	machineStates.stStartUp:
		Global.emgStop       := FALSE;
		Global.openDoors     := FALSE;
		Global.emgStopSignal := FALSE;
		resetSig             := FALSE;
		commandReady         := FALSE;
		purgeIndexDone       := FALSE;
		purgeRobotDone       := FALSE;
		purgeStackers		 := FALSE;
		Global.commands      := controlCommands.null;
		setDisplayState(machineDisplayStates.dStStartUp);
		NextState(machineStates.stInit);
	
//  *** Safety stop 
//  Има отворена врата, няма въздух или има натисната губа
//  Към всички станций се подава EMG сигнал

	machineStates.stSafetyStop:
		Global.commands      := controlCommands.null;
		Global.emgStopSignal := TRUE;
		resetTimer(IN := resetSig, PT := resetTime);
		
		IF      io.getX(ioImage.xDoors) 
			AND io.getX(ioImage.xAirOk) 
			AND io.getX(ioImage.xEmgBnt) 
			AND io.getX(ioImage.xRobotEmgOk)  THEN
				resetSig := TRUE;
				IF resetTimer.Q THEN	
					resetSig      := FALSE;
					nextState(machineStates.stInit);
				END_IF
		END_IF	

//  *** Init 
//  Инициализация на всички станций 
			
	machineStates.stInit:
		setDisplayState(machineDisplayStates.dStMachineStandBy);
		
		CASE Global.commands OF	
			controlCommands.start, 
			controlCommands.stop:
		        commandReady         := TRUE;
				Global.machError     := FALSE;
			    Global.emgStopSignal := FALSE;
			    nextState(machineStates.stReady);
				
			    Stations.incCommStBase.DoInit      := TRUE;			
			    Stations.sLoadStBase.DoInit        := TRUE;
				Stations.sUnloadStBase.DoInit      := TRUE;
				Stations.insertLoadStBase.DoInit   := TRUE;
				Stations.insertUnloadStBase.DoInit := TRUE;				
				Stations.roboStBase.DoInit         := TRUE;		
			
		END_CASE

// *** Ready 
// Синхронизира всички станций след подаване на захранването

	machineStates.stReady:
		depSync(Stations.incCommStBase,      globalDeps.depIncCommModeDone); 
		depSync(Stations.sLoadStBase,        globalDeps.depSLoadInit);
		depSync(Stations.sUnloadStBase,      globalDeps.depSUnloadInit);
		depSync(Stations.insertLoadStBase,   globalDeps.depILoadInitDone);
		depSync(Stations.insertUnloadStBase, globalDeps.depULoadInitDone);
		depSync(Stations.roboStBase,         globalDeps.depRoboInitDone);	
	
		nextState(machineStates.stCheckState);	
		
// *** Check state 
// В зависимост от зададената команда се задава следващо състояние

	machineStates.stCheckState:	
		IF NOT Global.purgeActive THEN	
			
			CASE Global.commands OF	
				controlCommands.start:
					nextState(machineStates.stAutoRun);
		   		controlCommands.stop:		
					nextState(machineStates.stStopping);
			END_CASE
			
		ELSE
			// Активна е purge процедура
			// Изчаква да се изпразни масата
			IF NOT purgeIndexDone THEN
				nextState(machineStates.stPurgeDialIndexSync);
			END_IF
			
			// Изчаква робота на приключи работа
			IF NOT purgeRobotDone THEN
				nextState(machineStates.stPurgeRobot);
			END_IF		

			// Изчаква стакерите да изкарат тарите в тях
			IF NOT purgeStackers THEN
				nextState(machineStates.stPurgeStackers);
			END_IF	
			
			nextState(machineStates.stPurgeDone);
			
		END_IF	

//  *** Stopping
//  Изчакват се всички станций да спрат

	machineStates.stStopping:
		setDisplayState(machineDisplayStates.dStMachineIsStopping);
		depSignal(globalDeps.depMachineStopping);
		depSync(Stations.incCommStBase,      globalDeps.depIncStop);		
		depSync(Stations.sLoadStBase,        globalDeps.depSLoadStop);
		depSync(Stations.sUnloadStBase,      globalDeps.depSUnloadStop);
		depSync(Stations.insertLoadStBase,   globalDeps.depILoadStop);
		depSync(Stations.insertUnloadStBase, globalDeps.depULoadStop);
		depSync(Stations.roboStBase,         globalDeps.depRoboStop);
		
		nextState(machineStates.stStopMach);
		
//  *** Stop 
//  Машината е спряна

	machineStates.stStopMach:	
		IF commandReady THEN
			Global.commands    := controlCommands.null;
			commandReady       := FALSE;	
		END_IF
	    setDisplayState(machineDisplayStates.dStMachineIsStopped);
	  
	    CASE Global.commands OF	
	      controlCommands.start:
		  	 commandReady := TRUE;
			 IF NOT Global.purgeActive THEN
		  		 nextState(machineStates.stAutoRun);	
			 ELSE
		  		 nextState(machineStates.stPurgeStart);
			 END_IF				 
							
		END_CASE	
	  
//  *** Auto run
//  Автоматичен режим

	machineStates.stAutoRun:
		IF commandReady THEN
			Global.commands    := controlCommands.null;
	    	commandReady       := FALSE;	
		END_IF
	    setDisplayState(machineDisplayStates.dStAutoRun);
		depSignal(globalDeps.depMachineAuto);
		IF Global.commands = controlCommands.stop THEN
		  	 commandReady := TRUE;				
		  	 nextState(machineStates.stStopping);			
		END_IF

// *** Purge - Start
// Изчистване на останалите в машита бройките
	
	machineStates.stPurgeStart:
		purgeIndexDone       := FALSE;
		purgeRobotDone       := FALSE;
		purgeStackers		 := FALSE;
		setDisplayState(machineDisplayStates.dStMachinePurgeActive);
		depSignal(globalDeps.depMachinePurgeStart);
		nextState(machineStates.stPurgeDialIndexSync);	
		
// *** Purge - Dial Index Sync
// Изчаква масата на InC да се завърти колкое необходимо пъти
// зада се изчистят останалите броки от нея
	
	machineStates.stPurgeDialIndexSync:	
		purgeIndexDone := FALSE;
		depSync(Stations.incCommStBase, globalDeps.depIncPurgeDone);
		nextState(machineStates.stPurgeRobot);		
		
// *** Purge - Robot Start
// Команда purge към робота
	
	machineStates.stPurgeRobot:	
		purgeIndexDone := TRUE;
		purgeRobotDone := FALSE;
		depSignal(globalDeps.depMachinePurgeRobot);
		depSync(Stations.roboStBase, globalDeps.depRoboPurgeDone);
		nextState(machineStates.stPurgeStackers);
		
// *** Purge - Stackers
// Команда purge към стакерите
	
	machineStates.stPurgeStackers:
		purgeRobotDone := TRUE;
		purgeStackers  := FALSE;	
		depSignal(globalDeps.depMacinePurgeStackers);	
		depSync(Stations.sLoadStBase,   globalDeps.depSLoadPurgeDone);	
		depSync(Stations.sUnloadStBase, globalDeps.depSUnloadPurgeDone);	
		nextState(machineStates.stPurgeDone);

// *** Purge - Done

	machineStates.stPurgeDone:	
		purgeStackers		 := TRUE;
		Global.purgeActive   := FALSE;
	    TagsHMI.startPurge   := FALSE;		
		nextState(machineStates.stStop);				
	
//  *** Machine error
//  В някоя станция има грешка

	machineStates.stMachError:
		Global.commands    := controlCommands.null;
		setDisplayState(machineDisplayStates.dStStationError);		
	
END_CASE

METHOD PRIVATE setEmg
VAR_INPUT
	
	emgOrAlarm				: Bool; 				// Дали метода е извикам за EMG stop или аларма

END_VAR

// Когато има EMG ситуация или аларма, се задава съответният state, 
// без оглед на текущото състояние на state машината.
// Аварийното спиратен е с по-голям приоритет от алармата

	stBase.DependencyState       := Consts.NO_DEPENDENCY;
	depActive                    := FALSE;
	syncActive                   := FALSE;
	statePass 			   		 := FALSE;
	depCount                     := 0;
	MEMSET(ADR(syncArr), 0, SIZEOF(syncArr));
	
	IF emgOrAlarm THEN
		stCurrentState               := machineStates.stSafetyStop;
		stBase.CurrentState          := machineStates.stSafetyStop;
	ELSE
		stCurrentState               := machineStates.stMachError;
		stBase.CurrentState          := machineStates.stMachError;
	END_IF
END_METHOD

ACTION zumer:
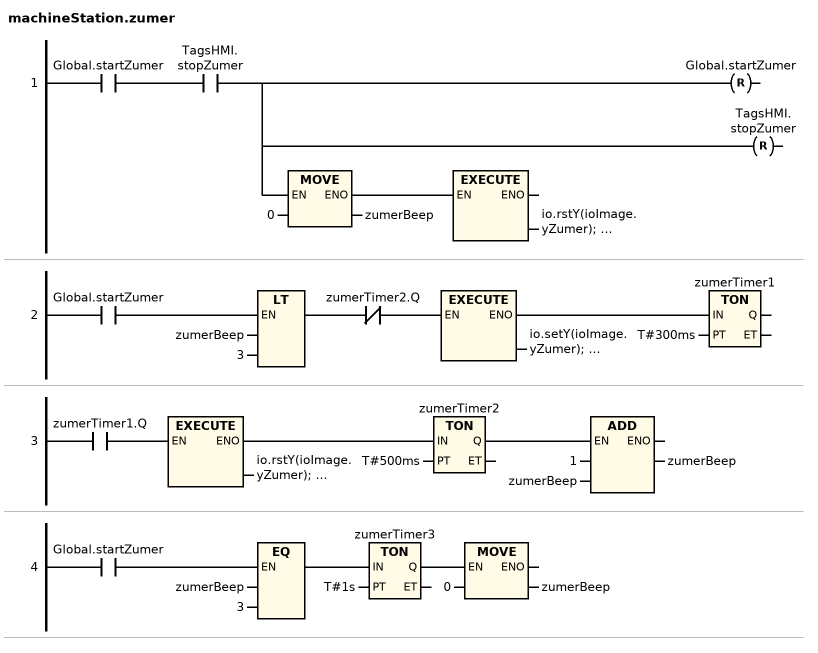
// NETWORK 1
_w1 := Global.startZumer AND TagsHMI.stopZumer;
Global.startZumer R= _w1;
TagsHMI.stopZumer R= _w1;
IF _w1 THEN zumerBeep := 0; END_IF
IF _w1 THEN io.rstY(ioImage.yZumer); END_IF

// NETWORK 2
_w2 := (Global.startZumer AND zumerBeep < 3) AND NOT zumerTimer2.Q;
IF _w2 THEN io.setY(ioImage.yZumer); END_IF
zumerTimer1(IN := _w2, PT := T#300ms); // TON

// NETWORK 3
_w3 := zumerTimer1.Q;
IF _w3 THEN io.rstY(ioImage.yZumer); END_IF
zumerTimer2(IN := _w3, PT := T#500ms); // TON
IF zumerTimer2.Q THEN zumerBeep := 1 + zumerBeep; END_IF

// NETWORK 4
zumerTimer3(IN := Global.startZumer AND zumerBeep = 3, PT := T#1s); // TON
IF zumerTimer3.Q THEN zumerBeep := 0; END_IF
END_ACTION

END_FUNCTION_BLOCK

// ---- POUs/stateMachine.TcPOU
FUNCTION_BLOCK stateMachine
VAR_INPUT

	stBase             : REFERENCE TO stationBase;	// Базова структура на станция  
	activeEMG          : BOOL;                      // Има активен safety стоп
	
	depClear           : BOOL;
	syncClear          : BOOL;

	
	
END_VAR
VAR_OUTPUT
END_VAR


VAR
	stCurrentState     : DINT;  			        // Текущо състояние на станцията
	startUp            : BOOL := FALSE;    		    // Флаг който се сетва за 1 цикъл при първо извикване 
	statePass		   : BOOL; 						// Вече има избран следващ state
	depPass            : BOOL; 						// Depandancy е било изпълнено за даденият state
	depSyncPass		   : BOOL;                    // Всички завицещи от текущият state, други станций са били sync-нати
	stationStop		   : BOOL; 				        // Станцията е спряна
	depActive          : BOOL;                      // Станцията изчаква друга
	syncActive         : BOOL;                      // Станцията sync-ва друга
	syncArr            : ARRAY [0..Consts.MAX_SYNC_STATIONS] OF INT; 
	depCount           : INT;                       // Общ брой на dependency-ta към други станий в текущият state
	depIndex           : INT;                       // Индек за адресиране на dependency в syncArr
	stTimer		       : TON;						// Всяки state има по един таймер
	stErrTimer         : TON;                       // И по един за генериране на грешка 
	startTimer         : BOOL;                      // Битове за старт на таймерите
	startErrTimer      : BOOL;
	stTime             : TIME;                      // Време на stTimer-a - задава се от stаteDalay
	stErrTime          : TIME;                      // Време за stErrТimer-a - задава се от timeOutError
	io				   : ioControl;                 // Дефинира няколко метода за работа с IO
	tempState          : DINT;                      // Запазва некущото състояни за step mode
	stepModeActive     : BOOL; 						// Активен е стъпков режим
	debugTimer         : TON;
	debugTImerIN       : BOOL;

END_VAR


// Тази част на FB-то никога няма да се изпълни (и кода в нея)

METHOD PRIVATE cycle
VAR_INPUT
	
	ioImage            : ANY;                           // ioImage за станцията 
	
END_VAR

VAR 
	ioImageIndex    : POINTER TO DINT;                 // показва началото на IO Image структурата
	ioStruct		: POINTER TO imageIO;              // текуща структура - една IO точка (DI или DO)
	points 			: DINT;							   // брой на входове и изходи в дадената стация
END_VAR

// Служи за упр. на стъпковата машина (в случея Switch Case блок)
// Грижи се за правилното упр. на сигнали от Staion Base

// Станцията е на автоматичен режим и е активна
IF stBase.AutoMode AND stBase.ToggleEnable THEN
	
	stBase.Disabled := FALSE;
	
	// Индекса за dependency-та се нулара всеки цикъл (изпползва се в dependencySync)
	depIndex        := 0;
		
	// При първо извикване станцията преминава в стартово състояние
	IF NOT startUp THEN
		startUp 			 	   	 := TRUE;
		stBase.Busy 	      	 	 := FALSE;
		stBase.Ready		 	 	 := FALSE;
		stBase.Error    	  		 := FALSE;
		stBase.LastState      		 := Consts.ST_START_UP;
		stBase.CurrentState   		 := Consts.ST_START_UP;
		stBase.Error          		 := FALSE;
		stBase.LastErrorState        := Consts.ST_NULL;
		stBase.DoInit         		 := FALSE;
		stBase.DoStart        		 := FALSE;
		stBase.DoStop        		 := FALSE;
		stBase.DependencyState       := Consts.NO_DEPENDENCY;	
		stCurrentState 				 := Consts.ST_START_UP;
		tempState 				     := Consts.ST_NULL;
		depCount 				     := 0;
		depActive                    := FALSE;
		syncActive                   := FALSE;
		statePass 			   		 := FALSE;
		depPass 				     := FALSE;
		depSyncPass 			     := FALSE;
		MEMSET(ADR(syncArr), 0, SIZEOF(syncArr));

	END_IF
	
	// Без оглед на текущото състояние се задава състояние на стоп
    // Ако има започанала някаква манупулация тя ще завърши 

	IF stBase.DoStop THEN
	
		stBase.DoStop             := FALSE;
		stationStop               := TRUE; 
		stBase.Busy 	      	  := FALSE;
		stBase.Ready		 	  := FALSE;
		stBase.Error              := FALSE;
		stepModeActive            := FALSE;
		depCount 				  := 0;
		depActive                 := FALSE;
		syncActive                := FALSE;
		statePass 			      := FALSE;
		depPass 				  := FALSE;
		depSyncPass 			  := FALSE;		
		stBase.CurrentState       := Consts.ST_STOP;
		tempState 				  := Consts.ST_NULL;
	
	END_IF
	
	// Когато станцията е спряла или е имало грешка при командта RESTART от HMI (DoInt)
	// станцията се инициализира
	IF  stBase.DoInit THEN
		
	    stBase.DoInit                := FALSE;
		stBase.Error                 := FALSE;
		stationStop    			     := FALSE;
		statePass 			   		 := FALSE;
		stBase.DoConfirmDependency   := FALSE;
		depCount 				     := 0;
		depActive                    := FALSE;
		syncActive                   := FALSE;
		statePass 			   		 := FALSE;
		depPass 				     := FALSE;
		depSyncPass 			     := FALSE;		
		stBase.DependencyState       := Consts.NO_DEPENDENCY;	
		stBase.LastErrorState        := Consts.ST_NULL;
		stBase.CurrentState          := Consts.ST_INIT;
        MEMSET(ADR(syncArr), 0, SIZEOF(syncArr));
	ELSE
		stBase.DoInit                := FALSE;
	END_IF
	
	// Има активен safety предпазен стоп
	IF activeEMG THEN
			
		stBase.DoConfirmDependency   := FALSE;
		statePass 			   		 := FALSE;
		depPass 				     := FALSE;
		depSyncPass 			     := FALSE;		
		depCount 				     := 0;
		depActive                    := FALSE;
		syncActive                   := FALSE;
		stBase.DependencyState       := Consts.NO_DEPENDENCY;
		stepModeActive     		     := FALSE;
		tempState 				     := Consts.ST_NULL;
		startTimer       		     := FALSE;
		startErrTimer                := FALSE;
		stBase.CurrentState          := Consts.ST_EMG;
		stCurrentState               := Consts.ST_EMG;
		MEMSET(ADR(syncArr), 0, SIZEOF(syncArr));
	
	END_IF
	
	IF NOT stBase.Error AND NOT stationStop THEN
		IF stCurrentState = Consts.ST_READY OR stCurrentState = Consts.ST_STEP_BLOCK THEN	
			stBase.Ready := TRUE;
			stBase.Busy  := FALSE;	
		ELSE
			stBase.Ready := FALSE;
			stBase.Busy  := TRUE;			
		END_IF
	ELSE
		stBase.Ready := FALSE;
		stBase.Busy  := FALSE;
	END_IF
	
	// Правене на преход от към ново състояние
	IF stCurrentState <> stBase.CurrentState THEN
		
		startTimer       := FALSE;
		startErrTimer    := FALSE;
		statePass 		 := FALSE;
		depPass 		 := FALSE;
		depSyncPass 	 := FALSE;
		
		stBase.DependencyState       := Consts.NO_DEPENDENCY;
		
		IF stBase.NextStep or stepModeActive THEN
			IF  stBase.CurrentState <> Consts.ST_STEP_BLOCK THEN
				stepModeActive       := TRUE;                 // Активен е спъпков режим
				stBase.NextStep      := FALSE;
				tempState            := stBase.CurrentState;
				stBase.CurrentState  := Consts.ST_STEP_BLOCK;
				stCurrentState       := Consts.ST_STEP_BLOCK;
			END_IF
		ELSE
			stBase.LastState := stCurrentState;
			stCurrentState   := stBase.CurrentState;        // Следващ state при автоматичрн режим
		END_IF
		
	END_IF
	
	IF stCurrentState = Consts.ST_STEP_BLOCK AND stBase.NextStep THEN
		stBase.CurrentState  := tempState; 	
		stCurrentState       := tempState;
		stBase.NextStep      := FALSE;	
		statePass 			 := FALSE;
		depPass 			 := FALSE;
		depSyncPass 	     := FALSE;		
	END_IF
	
	// При активен съпков режим може да се продължи към автоматичен
	IF stepModeActive AND stBase.DoStart THEN
		 stBase.CurrentState  := tempState; 	
		 stCurrentState       := tempState;
		 stBase.DoStart       := FALSE;
		 stepModeActive       := FALSE;	
		 statePass 			  := FALSE;	
		 depPass 			  := FALSE;
		 depSyncPass 		  := FALSE;		 
	END_IF

	
	// Таймери за state-та - един за общо ползване и един за ген. на грешка
	stTimer   (IN := startTimer,    PT := stTime);
	stErrTimer(IN := startErrTimer, PT := stErrTime);
	

    // Когато станцията е спяла тогава може да се сетват и ресетват входове и изходи
	// Чрез ANY pointer и малко аритметика се адресира структура по структура и се проверява
	// дали трябва да се сетне дадено IO 
	IF stationStop THEN

		points         := ioImage.diSize / SIZEOF(imageIO);     // брой IO points за станция
		ioImageIndex   := ioImage.pValue;                       // стартов адрес на структурата
	
		WHILE points > 0 DO                                     // адрес на imageIO 
			
			ioStruct := ioImageIndex;  
                         
			IF ioStruct^.iType = ioType.INPUT_BIT THEN          // updata на pointa ако е вход
				ioStruct^.stIO := io.getX(ioStruct^);
		
			ELSIF ioStruct^.iType = ioType.OUTPUT_BIT THEN	
				IF ioStruct^.stIO THEN
					io.setY(ioStruct^);
				ELSE 
					io.rstY(ioStruct^);
				END_IF
			END_IF
		
			ioImageIndex := ioImageIndex + SIZEOF(imageIO);      // dec -  следващ IO point
			points       := points - 1;
		END_WHILE
	END_IF
			
ELSE
	// Станцията е изключена
	stBase.Disabled := TRUE;	
	startUp         := TRUE;
	
END_IF
END_METHOD

METHOD PROTECTED depNextState
VAR_INPUT
	
	station			: REFERENCE TO stationBase;       
	dep 			: DINT;  
    newState 		: DINT;                                             

END_VAR


// Ако има сигнализарано dependency от depSignal, веднага се прави преход
// към зададеният state. Всички останли dependency-та, (ако имa) се изчистват
// Тоест тази метод е с по-висок приоритет от depSync и depWait

IF  station.DependencyState = dep AND stCurrentState = stBase.CurrentState THEN
	
	MEMSET(ADR(syncArr), 0, SIZEOF(syncArr));
	syncActive       := FALSE;
	depActive        := FALSE;
	nextState(newState);

END_IF
END_METHOD

METHOD PROTECTED depSignal
VAR_INPUT
		
	dep 		: DINT;	

END_VAR

// Сетва dependency, но не блокира на него какво в depWait.
// Отново има място само за едно на state.
// Изчиства се автоматично при преминаване в следващият state

IF stBase.DependencyState = Consts.NO_DEPENDENCY AND stCurrentState = stBase.CurrentState THEN
	stBase.DependencyState      := dep;
END_IF
END_METHOD

METHOD PROTECTED depSync
VAR_INPUT
	
	station			: REFERENCE TO stationBase;       // станция от която е извикан dependencyWait
	dep 			: DINT;                           // какво dependency е сетнато

// Трябва dependency-то което се очаква и това което sync-ва да са еднакви!
// Иначе ще има dead-lock в текущите състояние и на двете станций.                         


END_VAR

// Метода потвърждата дадето dependency от друга станция.
// В един state може да има до 64 Sync извиквания - докато всичките
// такива не се изпълнят станцията няма да мине в следващ state.

IF stCurrentState = stBase.CurrentState AND NOT depSyncPass THEN
	syncActive    := TRUE;                        // спира се възможноста за преход в друг state
	
	// Когато за първи път извика метода даденото dependency се макрира като вече отчетено
	// Брояча на dependency-та се увеличава. Така се знае колко трябва да се изпълнят за дадения state
	// и чак след като всички се sync-ват и може да се премине в следващ state
	IF syncArr[depIndex] = 0 THEN
	
		syncArr[depIndex] := Consts.DEP_PASS;
		depCount          := depCount + 1;

	// Има маркирано dependency и на него се чака в друга станция
	// Другата станция се "освобождава" а тук брояча на dependency-та се намалява - има sync-нато dependency
	ELSIF (syncArr[depIndex] = Consts.DEP_PASS AND station.DependencyState = dep) OR syncClear THEN
	
		syncArr[depIndex]       := Consts.SYNC_CONFIRM;
		station.DependencyState := Consts.NO_DEPENDENCY;
		depCount 		        := depCount - 1;
	
	END_IF
	
		depIndex          := depIndex + 1;
	
END_IF
END_METHOD

METHOD PROTECTED depWait

VAR_INPUT
	
     dep			: DINT;          // dependency което трябва да се Sync-не от друга станция

END_VAR

// Сетва определено dependency в stationBase
// Станцията не може да премине в друг state докато това dependency 
// не се потвърди от depenencySync ф-я.
// В един state може да има само едно извикване на dependencyWait, защото
// в stationBase има място само за едно.


IF stBase.DependencyState = Consts.NO_DEPENDENCY AND NOT depActive AND stCurrentState = stBase.CurrentState AND NOT depPass THEN
	stBase.DependencyState      := dep;
	depActive                   := TRUE;
ELSIF (stBase.DependencyState = Consts.NO_DEPENDENCY AND depActive) OR depClear THEN
	depActive 					:= FALSE;
	depClear                    := FALSE;
	depPass                     := TRUE;
END_IF
END_METHOD

METHOD PROTECTED nextState
VAR_INPUT
	
	nextState 		:DINT;                     // Следващо състояние

END_VAR

debugTimer(IN := debugTimerIN, PT := T#2S);

// Ако няма грешка или активно dependency или ако няма sync-ване

IF NOT stBase.Error AND NOT stationStop AND NOT depActive AND NOT syncActive AND NOT activeEMG AND NOT statePass THEN 

	IF DEBUG.noErrors THEN
		debugTimerIN := TRUE;
		IF debugTimer.Q THEN
		    stBase.CurrentState    := nextState;
			statePass 			   := TRUE;	
			debugTimerIN           := FALSE;
		END_IF	
	ELSE
  	    stBase.CurrentState    := nextState;
	    statePass 			   := TRUE;
	END_IF
	
END_IF
	

// При активно dependency, може да се премине в следващ state
// само ако брояча на dependency-та за дадения state e нула
// Това значи че те всички са sync-нати

IF syncActive AND depCount = 0  AND NOT depActive THEN

// Изчиства се масива в който е бил "маркиран" статута на 
// dependency-та в stata-та	

    MEMSET(ADR(syncArr), 0, SIZEOF(syncArr));
	
	syncActive             := FALSE;
    stBase.CurrentState    := nextState;
	statePass 			   := TRUE;
	depSyncPass            := TRUE;
		
END_IF
END_METHOD

METHOD PROTECTED setDisplayState
VAR_INPUT
	
	displayState		: DINT;         // състояние за виз. на HMI

END_VAR

// Просто актуализира променлива за displayState

IF displayState <> Consts.ST_NULL THEN
	stBase.DisplayState    := displayState;
END_IF
END_METHOD

METHOD PROTECTED setError
VAR_INPUT
		
	errState    :   DINT;       // състоянието за дадената грешка

END_VAR

// Този метод всъщност просто преминава към зададеното му състояние
// Разликата от nextState е че сетва и бит Error в stationBase
// Прехода се прави веднаги без да се отчита dependency 
IF NOT stBase.Error AND NOT stationStop AND stCurrentState = stBase.CurrentState AND NOT DEBUG.noErrors THEN 
	stBase.CurrentState    := errState;
	stBase.LastErrorState  := errState;
	stBase.Error           := TRUE;
    Global.machError       := TRUE;    

END_IF
END_METHOD

METHOD PROTECTED setStateVars
VAR_INPUT
	
    img            : ANY;       // ioImage за станцията 	

END_VAR
VAR_IN_OUT
	sv			: DINT; 		 // state var - текущо състояние
END_VAR

// Текущото състояние на станцията се записва като променлива 
// в stateMachine, за да могат всички методи да имат достъп до нея
// Изпълнява се упр. цикъл, update-ва се stateVar и се изпълнява главния switch case
// на станцията.

THIS^.stCurrentState := sv;

cycle(img);

sv := This^.stCurrentState;
END_METHOD

METHOD PROTECTED stateDelay : BOOL
VAR_INPUT

	t       : TIME;         // време на stTimer-a	

END_VAR

// Когато се извика тази ф-я стартира таймер
// Той е един за всяки state и е ощо ползване
// Min. времето е поне 10ms
// Ресетва се при преминаване в следващ state

IF t > T#10MS AND NOT startTimer THEN
	stTime     := t;
	startTimer := TRUE;	
END_IF


IF stTimer.Q THEN
	stateDelay   := TRUE;
ELSE
	stateDelay   := FALSE;
END_IF
END_METHOD

METHOD PROTECTED timeOutError
VAR_INPUT
	
	t				: TIME;      // време след което се ген. преминава в грешка
	stErr           : DINT;      // сътояние на грешката 

END_VAR
// Когато се извика тази ф-я стартира таймер
// След изтичането му се преминава в състояние не грешка
// Min. времето е поне 10ms
// Ресетва се при преминаване в следващ state

IF t > T#10MS AND NOT startErrTimer AND NOT DEBUG.noErrors THEN
	stErrTime       := t;
	startErrTimer   := TRUE;	
END_IF


IF stErrTimer.Q THEN
	setError(stErr);
END_IF
END_METHOD

END_FUNCTION_BLOCK

// ---- POUs/ioControl.TcPOU
FUNCTION_BLOCK ioControl
VAR_INPUT
END_VAR
VAR_OUTPUT
END_VAR
VAR
END_VAR


// Този блок има няколко метода който помагат за по-лесна работа на стъпковата машина
// 1. Метод за преминаване от състояние в състояние
// 2. Конфигурация на самата стъпкова машина
// 3. Няколко метода за четене и завпис на IO сигнали
// 4. State Taimer на базата на който да се генерира аларма

METHOD getSR : BOOL
VAR_INPUT

	xOn:  imageIO;      // Сигнал който трябва да е ON
    XOff: imageIO;      // Сигла който трябва да е OFF	

END_VAR

// Резултата се връща когато единият сигнал е ON, a другият ОFF
// Основно при друпозиционни устр.

IF getX(xOn) AND NOT getX(xOff) THEN
	getSR := TRUE;
ELSE
	getSR := FALSE;	
END_IF
END_METHOD

METHOD getX : BOOL

VAR_INPUT
	
		x	   : imageIO; 		// IO поле
		
END_VAR

VAR
	
		tempByte  : BYTE;
		mask      : BYTE;
		res       : BYTE;
		
END_VAR

// Прочита даден IO сигнал 

IF x.iType = ioType.INPUT_BIT THEN

	IF NOT DEBUG.ioDebugActive THEN	

		tempByte 		 := x.image^[x.iByte];       // Взима байта от IO Image
		mask     		 := SHL(1, x.iBit);         // Подготвя маската
  	 	 res              := tempByte AND mask;
		IF (res = 0) THEN
			getX   := FALSE;
			x.stIO := FALSE; 
		ELSE
			getX   := TRUE;
			x.stIO := TRUE; 
		END_IF
	ELSE	
		IF x.stIO THEN
			getX := TRUE;
		ELSE
			getX := FALSE;
		END_IF
	
	END_IF
	
END_IF
END_METHOD

METHOD rstY
VAR_INPUT
	
	y		: imageIO; 		// поле с IO изходен сигнал

END_VAR

VAR 
	  
	tempByte  : BYTE;
	mask      : BYTE;       // маска за сетване на опредене бит от байта
	
END_VAR
 // Ресетва изходен сигнал в периферията и в Station IO

 IF y.iType = ioType.OUTPUT_BIT THEN
	 
	IF NOT DEBUG.ioDebugActive THEN
	 
		y.stIO   		 := FALSE;         			//  Задава стойността в Station IO

		tempByte 		 := y.image^[y.iByte];       // Взима байта от IO Image
		mask     		 := SHL(1, y.iBit);         // Подготвя маската
		mask             := NOT mask; 				// Инвертирая
		y.image^[y.iByte] := tempByte AND mask;      // Ресетване на желаният бит
		
	ELSE
		y.stIO   		 := FALSE;         			//  Задава стойността в Station IO
END_IF
	
END_IF
END_METHOD

METHOD setSR
VAR_INPUT
	
	yOn:  imageIO;      // Изход който трябва да се сетне
    yOff: imageIO;      // Изход който трябва да се ресетне	

END_VAR

// Сетва първия и ресетва втория сигнал 
// За цилиндри основно

setY(yOn);
rstY(yOff);
END_METHOD

METHOD setY
VAR_INPUT
	
	y		: imageIO; 		// поле с IO изходен сигнал

END_VAR

VAR 
	  
	tempByte  : BYTE;
	mask      : BYTE;       // маска за сетване на опредене бит от байта
	
END_VAR

// Сетва изходен сигнал в периферията и в Station IO

IF y.iType = ioType.OUTPUT_BIT THEN
	
	IF NOT DEBUG.ioDebugActive THEN

		y.stIO           := TRUE;         			//  Задава стойността в Station IO
	
		tempByte 		 := y.image^[y.iByte];       // Взима байта от IO Image
		mask     		 := SHL(1, y.iBit);         // Подготвя маската
		y.image^[y.iByte] := tempByte OR mask;       // Сетване на желаният бит
		
	ELSE
		y.stIO           := TRUE;         			//  Задава стойността в Station IO
END_IF
	
END_IF
END_METHOD

END_FUNCTION_BLOCK

// ---- POUs/Stations/incCommStation.TcPOU
  FUNCTION_BLOCK incCommStation EXTENDS stateMachine
VAR_INPUT
	
	ioImage      		  : incCommImage;

END_VAR

VAR
	
	activeState            : incCommStates;	
	
	recipeTemp			   : DINT := 0;                       // Битова маска за рецепта на работа
	
	startPuls              	: R_TRIG;                         // Пулсов сигнал за START бутона
	stopPuls			   	: R_TRIG;                         // Пулсов сигнал за STOP бутона

	waitStationsReady       : BOOL := FALSE;                 // Изчаква станцийте са си завършат работата
	waitIndexReady		    : BOOL := FALSE; 				 // Изчаква индексирането на масата да завърши
	
	setModeDone			    : BOOL := FALSE; 				 // Има избран режим на работа
	purgeActive			    : BOOL := FALSE; 				 // PURGE процедурате е преключила
	purgeCycleCount		    : INT;                           // Брой завъртания при PURGE
	
END_VAR



// Натискането на бутони START и STOP на InC са извън цикъла на станицята.
// След натискането на бутон се сетва и съответната команда. Тя се изтрива при 
// аварийна ситуация или след като се изпълни в machine Station

startPuls(CLK := io.getX(ioImage.xSignalStart));
stopPuls (CLK := io.getX(ioImage.xSignalStop));	

IF Global.commands = controlCommands.null THEN
	
	IF startPuls.Q AND NOT stopPuls.Q THEN
		IF TagsHMI.startPurge THEN
			Global.commands     := controlCommands.start;
			Global.purgeActive  := TRUE;
		ELSE
			Global.commands     := controlCommands.start;				
		END_IF
	ELSIF stopPuls.Q  THEN 
		Global.commands    := controlCommands.stop;		
	END_IF
	
END_IF

// Има аларма в машината
IF Global.machError THEN
	io.setY(ioImage.yAlarm);
ELSE
	io.rstY(ioImage.yAlarm);	
END_IF


setStateVars(ioImage, activeState);

CASE activeState OF 
	
// *** Start Up 

	incCommStates.stStartUp:
		setDisplayState(incCommDisplayStates.dStStartingUp);
		Global.commands     := controlCommands.null;
		Global.sensorStatus := FALSE;
		setModeDone         := FALSE;
		purgeActive 	    := FALSE;
		waitIndexReady      := FALSE;
		waitStationsReady   := FALSE;
		recipeTemp          := 0;
		Global.recipe       := 0;
		io.rstY(ioImage.yDailIndex);
		io.setY(ioImage.yProductChange);                   // Разрешава избора на нов режим и лот в InC MMI		
		nextState(incCommStates.stInit);

// *** Init  

	incCommStates.stInit:

		IF NOT setModeDone AND NOT Global.purgeActive THEN
			nextState(incCommStates.stSetMode);
		ELSE
			nextState(incCommStates.stReady);
		END_IF
	
// *** Set Mode  - Тук се избира вида на режима на работа: HEX24 или HEX27

	incCommStates.stSetMode:	
    	setDisplayState(incCommDisplayStates.dStStandBy);	
		io.setY(ioImage.yProductChange);                   // Разрешава избора на нов режим и лот в InC MMI
	
		IF Global.commands = controlCommands.start THEN
			
			IF io.getX(ioImage.xRecipeBit0) THEN
				recipeTemp.0 := TRUE;
			ELSE
				recipeTemp.0 := FALSE;
			END_IF	
			
			IF io.getX(ioImage.xRecipeBit1) THEN
				recipeTemp.1 := TRUE;
			ELSE
				recipeTemp.1 := FALSE;
			END_IF	
	
			IF io.getX(ioImage.xRecipeBit2) THEN
				recipeTemp.2 := TRUE;
			ELSE
				recipeTemp.2 := FALSE;
			END_IF		
		
			IF io.getX(ioImage.xRecipeBit3) THEN
				recipeTemp.3 := TRUE;
			ELSE
				recipeTemp.3 := FALSE;
			END_IF		
				
			IF recipeTemp > 0 AND recipeTemp <= Consts.MAX_RECIPE THEN 
				Global.recipe   := recipeTemp;
				recipeTemp      := 0;
				setModeDone     := TRUE;
				nextState(incCommStates.stReady);
			ELSE
				setError(incCommStates.stErrCommFault);	
				recipeTemp      := 0;				
			END_IF			
		
		END_IF	
		
// *** Ready - Има избран режим и станцията се sync с machine station

	incCommStates.stReady:
		io.rstY(ioImage.yProductChange);
		depNextState(stations.machineStBase, GlobalDeps.depMachineStop,     incCommStates.stStationStop);	
		depNextState(stations.machineStBase, GlobalDeps.depMachineStopping, incCommStates.stStationStop);	
		depWait(globalDeps.depIncCommModeDone);
		
		IF Global.purgeActive AND NOT purgeActive THEN
			nextState(incCommStates.stStationStop);		
		END_IF
		
		IF NOT waitStationsReady THEN
			nextState(incCommStates.stIndexStart);
		END_IF
		
		IF NOT waitIndexReady THEN
			nextState(incCommStates.stIndexStationsReady);
		END_IF
		
// *** Stopped
// Станцията е спряна - може да с стартира или да се избере PURGE 

	incCommStates.stStationStop:
        setDisplayState(incCommDisplayStates.dStStationIsStopped);	
		io.rstY(ioImage.yDailIndex);
		io.rstY(ioImage.yProductChange);
		depWait(GlobalDeps.depIncStop);	
		depNextState(stations.machineStBase, GlobalDeps.depMachineAuto,       incCommStates.stIndexStart);
		depNextState(stations.machineStBase, GlobalDeps.depMachinePurgeStart, incCommStates.stPurgeStart);		

// *** Index - Start 

	incCommStates.stIndexStart:
		depNextState(stations.machineStBase, GlobalDeps.depMachineStop,     incCommStates.stStationStop);	
		depNextState(stations.machineStBase, GlobalDeps.depMachineStopping, incCommStates.stStationStop);
		IF NOT setModeDone THEN               // След PURGE трябва да се зададе нова рецепта
			setError(incCommStates.stErrCommFault);	
		ELSE
			waitStationsReady := FALSE;
			setDisplayState(incCommDisplayStates.dStWaitForAllStatinsReady);
			nextState(incCommStates.stIndexEnableStations);
	    END_IF		
						
// *** Index -  Enable Stations
// Дава се разрешение на всики станий да започнат работа

	incCommStates.stIndexEnableStations:
		IF io.getX(ioImage.xPickNestLoaded) THEN
			Global.sensorStatus := TRUE;
		ELSE
			Global.sensorStatus := FALSE;
		END_IF	
		IF NOT Global.robotSafe OR Global.commands = controlCommands.stop THEN  // Спира масата да се завърти при първо пускане на машината
			depSync(Stations.insertLoadStBase,   globalDeps.depILoadWaitIndex);
			depSync(Stations.insertUnloadStBase, globalDeps.depULoadWaitIndex);
			nextState(incCommStates.stIndexStationsReady);
		END_IF
		
// *** Index - Stations Ready
// Всички стаций който зависят от масата трябва да са готови преди тя да направи ход

	incCommStates.stIndexStationsReady:		
		waitStationsReady := TRUE;
		waitIndexReady    := FALSE;	
		depSync(Stations.insertLoadStBase,   globalDeps.depILoadDone);
		depSync(Stations.insertUnloadStBase, globalDeps.depULoadDone);		
		nextState(incCommStates.stSignalStations);
		
// *** Index - Singla Stations
// Цъкъла е завършен - може да се върти масата

	incCommStates.stSignalStations:	
		depSignal(globalDeps.depIncCycleDone);
		nextState(incCommStates.stIndexEnable);	
		
// *** Index -  Enable
// Дава се разрешение InC да завърди масата си

	incCommStates.stIndexEnable:		
		setDisplayState(incCommDisplayStates.dStDialTableIndexPermition);
		io.setY(ioImage.yDailIndex);
		IF NOT io.getX(ioImage.xDailIndexDone) THEN
			nextState(incCommStates.stIndexReady);
		END_IF
		
// *** Index -  Ready
// Масата се е завъртяла с 1 ход и е приключила хода си

	incCommStates.stIndexReady:	
		IF io.getX(ioImage.xDailIndexDone) THEN
			io.rstY(ioImage.yDailIndex);
			nextState(incCommStates.stIndexCheck);
			IF purgeActive THEN
				purgeCycleCount := purgeCycleCount + 1;
			END_IF
		END_IF	

// *** Index - Check
// Проверка дали цикъла е завършил или е активка PURGE процедура

	incCommStates.stIndexCheck:
		IF purgeActive AND purgeCycleCount = Consts.PURGE_CYCLES THEN
			nextState(incCommStates.stPurgeFinish);
		ELSE
			nextState(incCommStates.stIndexDone);
		END_IF			
	
// *** Index - Done

	incCommStates.stIndexDone:	
		waitIndexReady := TRUE;
		setDisplayState(incCommDisplayStates.dStDialTableIndexReady);
		nextState(incCommStates.stIndexStart);
		
// *** Purge - Start
// Стартира процедура PURGE като започва да брой колко завъртания е направила масата

	incCommStates.stPurgeStart:			
		purgeCycleCount := 0;
		purgeActive     := TRUE;
		nextState(incCommStates.stIndexStart);
		
// *** Purge - Finish
// Масата е направила необходимияят брой завъртания, сега се изчакват и другите 
// станций на машината да приключат с PURGE

	incCommStates.stPurgeFinish:	
		depWait(globalDeps.depIncPurgeDone);
		nextState(incCommStates.stPurgeDone);

// *** Purge - Done

	incCommStates.stPurgeDone:
		purgeActive        := FALSE;
		waitIndexReady     := FALSE;
		waitStationsReady  := FALSE;
		setModeDone        := FALSE;
		Global.purgeDoneIL := TRUE;
		Global.purgeDoneIU := TRUE;		
		Global.recipe      := 0;		
		nextState(incCommStates.stStationStop);

// *** ERROR  -  Има проблем със сигналите за избор на режим от InC
	
	incCommStates.stErrCommFault:
		setDisplayState(incCommDisplayStates.dStIncModeSignalsError);
		io.rstY(ioImage.yProductChange);
		io.rstY(ioImage.yDailIndex);

// *** EMG state - реално тук EMG стате не прави нищо освен да изчисти текущата команда

	incCommStates.stEMG:
		io.rstY(ioImage.yDailIndex);
		nextState(incCommStates.stInit);
		
// *** STOP
// Станцията е деактивирана

	incCommStates.stStop:
		waitStationsReady := FALSE;
		waitIndexReady    := FALSE;
	
// *** Step mode
// Скъпков режим на станцията

	incCommStates.stStepBlock:
		setDisplayState(incCommDisplayStates.dStWaitForNextStep);	
	

END_CASE

END_FUNCTION_BLOCK

// ---- POUs/Stations/stackerLoadStation.TcPOU
FUNCTION_BLOCK stackerLoadStation EXTENDS stateMachine

VAR_INPUT
	
	ioImage                : stackerLoadImage;

END_VAR

VAR

	activeState            : stackerLoadStates;	
	axisFesto              : FB_FESTO_CMMT_AS;
	
	resetDone			   : BOOL := FALSE; 						   // Стакера е в горна позиция и очаква зареждане
	palletsLoadDone		   : BOOL := FALSE;							   // Операта е заредил тари в стакера
	preparePalletDone      : BOOL := FALSE; 						   // Стакера зарежда тара
	moveDownDone		   : BOOL := FALSE;							   // Стакера е заредил тара и дрябва да се мръдне 1 ход надолу
	palletReleaseStart	   : BOOL := FALSE; 						   // Има взета тара от върха на стакера	
	purgeStart			   : BOOL := FALSE; 						   // Процедура за изпразване на стакера    
	roboOutStart           : BOOL := FALSE;                            // Робота трябва да е надалеч, че да се зарежда нова тара	
	moveDone		       : BOOL := FALSE; 						   // Фесто мотора си е изпълнил заданието при движение	
	
	posCount			   : DINT;					 				   // Брой позиций на оста
	axisLen				   : REAL;				
	currentPos 			   : DINT;					 				   // Текуща позиция
	axisPosArr			   : ARRAY [0..Consts.MAX_AXIS_POS] OF REAL;   // Масив с позицийте на оста

	cylinderTimeOut		   : TIME := T#2S;                             // Време за ход на цилиндър
	driveEnTime		       : TIME := T#1S;							   // Време за enable на фесто drive
	initMoveTimeOut		   : TIME := T#20S;                            // Време за ход до крайно горно положение
	sensorTime 			   : TIME := T#250MS;                          // Време за реакция на оптичен сензор
	palletsLoadTimeOut	   : TIME := T#15S; 						   // Време за ход на зареждане на тари
	palletMoveTimeOut	   : TIME := T#10S;                            // Време за преместване на 1 позиция
	drivePosTime           : TIME := T#100MS;                          // Време за задаване на задание за позициониране	

END_VAR


drivesControl();          // Упр. на Феесто мотора дрижещ осна на стакера

setStateVars(ioImage, activeState);


CASE activeState OF 
	
//  *** Start Up
//  Старт на станцията след подаване на захр.	

	stackerLoadStates.stStartUp:
		setDisplayState(stackerLoadDisplayStates.dStStartingUp);
		Stations.sLoadDrive.DoEnable  := FALSE;
		Stations.sLoadDrive.DoMove    := FALSE;						   						   
		nextState(stackerLoadStates.stPowerUp);
		
//  *** Power Up - Start
//  Инициализация след подaване на захранване

	stackerLoadStates.stPowerUp:
		IF io.getX(ioImage.xPalletOnTop) THEN
			setError(stackerLoadStates.stErrRemovePallet);
		END_IF
		
//  *** Init 
//  Инициализация на станцията
	
	stackerLoadStates.stInit:
	
		depWait(globalDeps.depSLoadInit);		

		// Проверка за приключила инициализация - стакера е горе, празен
		IF NOT resetDone THEN
			nextState(stackerLoadStates.stResetStart);
	    END_IF	
		
		// Проверка за приключило зареждане на тари - стакера е пълен 
		IF NOT palletsLoadDone THEN
			nextState(stackerLoadStates.stLoadPalletsStart);		
		END_IF
		
		// Проверка за приключило зарездане на тара - има заредена тара на върха на стакера
		IF NOT preparePalletDone THEN
			nextState(stackerLoadStates.stPreparePalletStart);		
		END_IF
		
		// Проверка дали след като е заредила тара, стакера се е преместил 1 ход надолу
		IF NOT moveDownDone THEN
			nextState(stackerLoadStates.stMoveDownStart);
		END_IF
		
		// Робото е готов да вземе вече празната тара
		IF  palletReleaseStart THEN
			nextState(stackerLoadStates.stReleasePalletStart);
		END_IF
		
		// Робото трябва да се отдаличил 
		IF  roboOutStart THEN
			nextState(stackerLoadStates.stRoboOutStart);
		END_IF		
		
		// Проверява дали е приключила PURGE  процедура
		IF purgeStart THEN
			nextState(stackerLoadStates.stLoadPurgeStart);
		END_IF
		
		nextState(stackerLoadStates.stInitDone);
		
// *** Init Done
// След излизането от аварийна ситуация или след изчисването на грешка
// станция е завършила своята инициализация

	stackerLoadStates.stInitDone:
		IF io.getX(ioImage.xPalletOnTop) THEN
			nextState(stackerLoadStates.stReady);
		ELSIF stateDelay(sensorTime * 2) AND NOT io.getX(ioImage.xPalletOnTop) THEN
			nextState(stackerLoadStates.stPreparePalletStart);
			preparePalletDone  := FALSE;		
		END_IF	
				
// *** Ready
// Станцията е готова за работа и очаква команда от machine
// Или робота е готов да вземе празната вече тара

	stackerLoadStates.stReady:
		setDisplayState(stackerLoadDisplayStates.dStStandBy);
		depNextState(Stations.machineStBase, GlobalDeps.depMachineStopping,     stackerLoadStates.stStackerStopped);
		depNextState(Stations.machineStBase, GlobalDeps.depMachineStop,         stackerLoadStates.stStackerStopped);		
	    depNextState(Stations.machineStBase, GlobalDeps.depMacinePurgeStackers, stackerLoadStates.stLoadPurgeStart);	
	    depNextState(Stations.roboStBase,    GlobalDeps.depSLoadRobotLoadGrip,  stackerLoadStates.stReleasePalletStart);			
		
// *** Stacker is Stopped
// Стакера е спрял след като е завършил текущият си цикъл и е бил натиснат STOP бутона
	stackerLoadStates.stStackerStopped:
        setDisplayState(stackerLoadDisplayStates.dStStationIsStopped);	
		Stations.sLoadDrive.DoMove       := FALSE;
		Stations.sLoadDrive.DoEnable     := FALSE;
		depWait(GlobalDeps.depSLoadStop);	
		depNextState(stations.machineStBase, GlobalDeps.depMachineAuto,       stackerLoadStates.stInitDone);
		depNextState(stations.machineStBase, GlobalDeps.depMachinePurgeStart, stackerLoadStates.stReady);
		
// *** Reset - Start
// Започва инициялизация на стакера - трябва да се премести 
// нагоре докрай. Затова първо робота трябва да е на безопасно място.	

	stackerLoadStates.stResetStart:
		resetDone   := FALSE;
		setDisplayState(stackerLoadDisplayStates.dStStackerIsReseting);
		IF NOT Global.robotSafe THEN
			depWait(globalDeps.depSLoadWaitRobotReady);
			nextState(stackerLoadStates.stResetUnlockPallet);			
		ELSE
			nextState(stackerLoadStates.stResetUnlockPallet);			
		END_IF

// ***  Reset - Unlock Pallet
// Всички ключалки на стакера се отварят

	stackerLoadStates.stResetUnlockPallet:
		io.setSR(ioImage.yLocks_unlock, ioImage.yLocks_lock);
		io.setSR(ioImage.yPalletFix_unlock, ioImage.yPalletFix_lock);
		nextState(stackerLoadStates.stResetCheckLocks);	

// *** Reset - Check Locks
// Проверка дали всички ключалки да се отворили

	stackerLoadStates.stResetCheckLocks:
		IF io.getSR(ioImage.xLock1_unlock, ioImage.xLock1_lock) AND 
		   io.getSR(ioImage.xLock2_unlock, ioImage.xLock2_lock) AND
		   io.getSR(ioImage.xPalletFix_unlock, ioImage.xPalletFix_lock) THEN
		   		nextState(stackerLoadStates.stResetEnableDrive);
		END_IF
		
		IF stateDelay(cylinderTimeOut) THEN
			
			IF NOT io.getSR(ioImage.xLock1_unlock, ioImage.xLock1_lock) THEN
				setError(stackerLoadStates.stErrLock1NotOpen);
			ELSIF NOT io.getSR(ioImage.xLock2_unlock, ioImage.xLock2_lock) THEN
				setError(stackerLoadStates.stErrLock2NotOpen);
			ELSIF NOT io.getSR(ioImage.xPalletFix_unlock, ioImage.xPalletFix_lock) THEN
				setError(stackerLoadStates.stErrFixerNotOpen);
		    END_IF
			
		END_IF 

// *** Reset - Enable Drive
// Enable на фесто мотора

	stackerLoadStates.stResetEnableDrive:
		IF Stations.sLoadDrive.Error THEN
			Stations.sLoadDrive.DoReset  := TRUE;
		ELSE
			Stations.sLoadDrive.DoReset  := FALSE;
			Stations.sLoadDrive.DoEnable := TRUE;
			IF stateDelay(driveEnTime) THEN
				nextState(stackerLoadStates.stResetDriveMove);
			END_IF
		END_IF
		timeOutError(driveEnTime*2, stackerLoadStates.stErrAxis);

// *** Reset - Init Drive
// Премества стакера в горно положение

	stackerLoadStates.stResetDriveMove:
		IF Stations.sLoadDrive.Enabled AND NOT Stations.sLoadDrive.Error THEN
			Stations.sLoadDrive.TargetPosition     := Stations.sLoadSettings.pallet[Global.recipe].zeroPos;
			Stations.sLoadDrive.TargetAcceleration := Stations.sLoadSettings.axisAcc;
			Stations.sLoadDrive.TargetVelocity     := Stations.sLoadSettings.axisInitSpeed;
			Stations.sLoadDrive.DoMove             := TRUE;
			moveDone							   := FALSE;
			IF stateDelay(drivePosTime) THEN
				nextState(stackerLoadStates.stResetCheckDrive);
			END_IF	
		ELSE
			setError(stackerLoadStates.stErrAxis);
	   END_IF
	   
// *** Reset - Check Drive
// Проверка дали е завършил хода на оста  

	stackerLoadStates.stResetCheckDrive:
		IF Stations.sLoadDrive.TargetReached AND NOT Stations.sLoadDrive.Error THEN
			Stations.sLoadDrive.DoMove := FALSE;
			moveDone 				   := TRUE;
			nextState(stackerLoadStates.stResetDone);	
		ELSIF NOT Stations.sLoadDrive.TargetReached AND Stations.sLoadDrive.Error THEN
			setError(stackerLoadStates.stInitMoveErr);
		END_IF	
		timeOutError(initMoveTimeOut, stackerLoadStates.stInitMoveErr);
		
//  *** Reset - Done
// Началната инициализация е приключила.
// Изчаква се оператора да зареди тарите - затова трябва да отвори врата (stEMG)
		
	stackerLoadStates.stResetDone:
		setDisplayState(stackerLoadDisplayStates.dStWaitForPalletsLoading);		
		IF NOT purgeStart THEN
			resetDone       		  := TRUE;
        	palletsLoadDone           := FALSE;
			TagsHMI.LoadStackerSignal := TRUE;
		ELSE	
			nextState(stackerLoadStates.stLoadPurgeConfirm);
		END_IF		

// *** Purge - Confirm
// Този state се изпълнява само при край на PURGE - за може правилно да завърши тази процедура

	stackerLoadStates.stLoadPurgeConfirm:
		 purgeStart                := FALSE;	
		 resetDone                 := TRUE;
         palletsLoadDone           := FALSE;		
		 TagsHMI.LoadStackerSignal := TRUE;	 
		 depWait(globalDeps.depSLoadPurgeDone);
	
// *** Pallets Load - Start
// Трябва да се заредят поставените от оператора тари в стакера

	stackerLoadStates.stLoadPalletsStart:
		palletsLoadDone   := FALSE;
		setDisplayState(stackerLoadDisplayStates.dStLoadPallets);
		nextState(stackerLoadStates.stPalletsLoadLimitCheck);
		
//  *** Pallets Load - Limit check
//  Проверяват се дали има зададени параметри на хода на стакера
//  Ако няма такива НЕ може да се продължи с инизиализацията		
		
	stackerLoadStates.stPalletsLoadLimitCheck:
		IF Stations.sLoadSettings.axisLength < Consts.MIN_AXIS_LEN OR Stations.sLoadSettings.pallet[Global.recipe].size < Consts.MIN_PALLET_SIZE THEN
			setError(stackerLoadStates.stErrNoProperSettings);
		END_IF
		nextState(stackerLoadStates.stPalletsLoadCalcAxis);	

//  *** Pallets Load -  Calc Axis
//  Изчисляват се позицийте за хода на оста на стакера 	
		
	stackerLoadStates.stPalletsLoadCalcAxis:    
	    axisLen       := Stations.sLoadSettings.pallet[Global.recipe].zeroPos;
		axisPosArr[0] := Stations.sLoadSettings.pallet[Global.recipe].zeroPos;
		currentPos 	  := 1;
		posCount      := 1;
		
		WHILE axisLen < Stations.sLoadSettings.axisLength AND currentPos < Consts.MAX_AXIS_POS DO
			axisLen    			   := axisLen + Stations.sLoadSettings.pallet[Global.recipe].size;
			axisPosArr[currentPos] := axisLen;
			currentPos  := currentPos + 1;
		END_WHILE
		
		posCount     := currentPos;
		currentPos   := 0;
		nextState(stackerLoadStates.stPalletsLoadCheckTop);
		
// *** Load Pallets - Check Top
// Oтварят се всички ключалки

	stackerLoadStates.stPalletsLoadCheckTop:
		io.setSR(ioImage.yLocks_unlock, ioImage.yLocks_lock);
		io.setSR(ioImage.yPalletFix_unlock, ioImage.yPalletFix_lock);
		nextState(stackerLoadStates.stPalletsLoadCheckLocks);
	
		
// *** Load Pallets - Check Locks
// Проверка, че всички ключалки са се отворили 

	stackerLoadStates.stPalletsLoadCheckLocks:
		IF io.getSR(ioImage.xLock1_unlock, ioImage.xLock1_lock) AND 
		   io.getSR(ioImage.xLock2_unlock, ioImage.xLock2_lock) AND
		   io.getSR(ioImage.xPalletFix_unlock, ioImage.xPalletFix_lock) THEN
		   		nextState(stackerLoadStates.stLoadPalletsDriveOn);
		END_IF
		
		IF stateDelay(cylinderTimeOut) THEN
			
			IF NOT io.getSR(ioImage.xLock1_unlock, ioImage.xLock1_lock) THEN
				setError(stackerLoadStates.stErrLock1NotOpen);
			ELSIF NOT io.getSR(ioImage.xLock2_unlock, ioImage.xLock2_lock) THEN
				setError(stackerLoadStates.stErrLock2NotOpen);
			ELSIF NOT io.getSR(ioImage.xPalletFix_unlock, ioImage.xPalletFix_lock) THEN
				setError(stackerLoadStates.stErrFixerNotOpen);
		    END_IF
		END_IF
		
//  *** Load Pallets - Drive On 
// Проверява дали всичко е наред с мотора

	stackerLoadStates.stLoadPalletsDriveOn:
		IF Stations.sLoadDrive.Error THEN
			Stations.sLoadDrive.DoReset  := TRUE;
		ELSE
			Stations.sLoadDrive.DoReset  := FALSE;
			Stations.sLoadDrive.DoEnable := TRUE;
			IF stateDelay(driveEnTime) THEN
				setDisplayState(stackerLoadDisplayStates.dStLoadPallets);
				nextState(stackerLoadStates.stLoadPalletsCalcPos);
			END_IF
		END_IF
		timeOutError(driveEnTime * 2, stackerLoadStates.stErrAxis);	
		
//  *** Load Pallets  - Calc Pos
// Изчислява следващата позиция 
// Стакера слиза надолу с определен брой тари - така, ако оператора не е заредил
// max. брой тази не се изчаква много после при движениет нагоре
	
		
	stackerLoadStates.stLoadPalletsCalcPos:
		IF currentPos = posCount AND moveDone THEN
			nextState(stackerLoadStates.stLoadPalletsMoveAgain);
		ELSIF moveDone THEN
			currentPos     := currentPos  + Consts.LOAD_PALLETS_STEP;
			IF currentPos >= posCount THEN
				currentPos := posCount;
			END_IF
		END_IF
		Stations.sLoadDrive.TargetPosition     := axisPosArr[currentPos];
		Stations.sLoadDrive.TargetAcceleration := Stations.sLoadSettings.axisAcc;
		Stations.sLoadDrive.TargetVelocity     := Stations.sLoadSettings.axisWorkSpeed;
		Stations.sLoadDrive.DoMove             := TRUE;
		moveDone						       := FALSE;
		IF stateDelay(drivePosTime) THEN
			nextState(stackerLoadStates.stLoadPalletsMoveDone);
		END_IF	
		
//  *** Load Pallets -  Move Done
// Стакера е направил хода си 

	stackerLoadStates.stLoadPalletsMoveDone:
		IF Stations.sLoadDrive.TargetReached AND NOT Stations.sLoadDrive.Error THEN
			Stations.sLoadDrive.DoMove := FALSE;
			moveDone			       := TRUE;
			nextState(stackerLoadStates.stLoadPalletsMoveAgain);	
		ELSIF NOT Stations.sLoadDrive.TargetReached AND Stations.sLoadDrive.Error THEN
			setError(stackerLoadStates.stErrPalletLoad);
		END_IF	
		timeOutError(palletsLoadTimeOut, stackerLoadStates.stErrPalletLoad);	
		
//  *** Load Pallets - Move again
// Проверка дали стакера да продължи надолу или е заредил тарите

	stackerLoadStates.stLoadPalletsMoveAgain:
		IF io.getX(ioImage.xPalletOnTop) AND currentPos <> posCount THEN
			nextState(stackerLoadStates.stLoadPalletsCalcPos);
		ELSIF io.getX(ioImage.xPalletOnTop) AND currentPos = posCount THEN
			setError(stackerLoadStates.stErrRemovePallet);			
		END_IF
		IF stateDelay(sensorTime * 2) THEN
			nextState(stackerLoadStates.stLoadPalletsDone);			
		END_IF
		
// *** Pallets Load - Done
// Всички тари са заредени

	stackerLoadStates.stLoadPalletsDone:
		palletsLoadDone := TRUE;	
		nextState(stackerLoadStates.stPreparePalletStart);
		
// *** Prepare Pallet - Start
// Стакера започва да се предвижва по 1 стъпка нагоре докато детектне тара

	stackerLoadStates.stPreparePalletStart:
		preparePalletDone := FALSE;
		setDisplayState(stackerLoadDisplayStates.dStWaitForPallet);	
		nextState(stackerLoadStates.stPreparePalletCheckTop);

// ***  Prepare Pallet - Check Top
//  Отваряне на всички грипери

	stackerLoadStates.stPreparePalletCheckTop:
		io.setSR(ioImage.yLocks_unlock, ioImage.yLocks_lock);
		io.setSR(ioImage.yPalletFix_unlock, ioImage.yPalletFix_lock);
		nextState(stackerLoadStates.stPreparePalletCheckLocks1);

// *** Prepare Pallet - Check Locks
// Проверка, че всички ключалки са се отворили 

	stackerLoadStates.stPreparePalletCheckLocks1:
		IF io.getSR(ioImage.xLock1_unlock, ioImage.xLock1_lock) AND 
		   io.getSR(ioImage.xLock2_unlock, ioImage.xLock2_lock) AND
		   io.getSR(ioImage.xPalletFix_unlock, ioImage.xPalletFix_lock) THEN
		   		nextState(stackerLoadStates.stPreparePalletSyncRobot);
		END_IF
		
		IF stateDelay(cylinderTimeOut) THEN
			
			IF NOT io.getSR(ioImage.xLock1_unlock, ioImage.xLock1_lock) THEN
				setError(stackerLoadStates.stErrLock1NotOpen);
			ELSIF NOT io.getSR(ioImage.xLock2_unlock, ioImage.xLock2_lock) THEN
				setError(stackerLoadStates.stErrLock2NotOpen);
			ELSIF NOT io.getSR(ioImage.xPalletFix_unlock, ioImage.xPalletFix_lock) THEN
				setError(stackerLoadStates.stErrFixerNotOpen);
		    END_IF
		END_IF		
		
// *** Prapare Pallet - Sync Robot
// Робота трябва да е на безопастно място за се движи стакета нагоре

	stackerLoadStates.stPreparePalletSyncRobot:
		IF Stations.sLoadDrive.Enabled AND NOT Stations.sLoadDrive.Error THEN
			nextState(stackerLoadStates.stPreparePalletMove);
		ELSE
			nextState(stackerLoadStates.stPrepareDriveOn);			
		END_IF		
			
//  *** Prapare Pallet - Drive On
// Активира се мотора на оста за да направи 1 ход нагоре

	stackerLoadStates.stPrepareDriveOn:
		IF Stations.sLoadDrive.Error THEN
			Stations.sLoadDrive.DoReset  := TRUE;
		ELSE
			Stations.sLoadDrive.DoReset  := FALSE;
			Stations.sLoadDrive.DoEnable := TRUE;
			IF stateDelay(driveEnTime) AND Stations.sLoadDrive.Enabled THEN
				setDisplayState(stackerLoadDisplayStates.dStWaitForPallet);
				nextState(stackerLoadStates.stPreparePalletMove);
			END_IF
		END_IF
		timeOutError(driveEnTime * 2, stackerLoadStates.stErrAxis);	
			
// *** Prapare Pallet - Move Up 
// Прества стакера нагоре с 1 поз.

	stackerLoadStates.stPreparePalletMove:
		IF moveDone THEN
			currentPos := currentPos - 1;
		END_IF
		IF currentPos < 0 THEN
			currentPos           := 0;
			palletsLoadDone      := FALSE;
			Global.startZumer    := TRUE;
			Global.lStackerEmpty := TRUE;
			nextState(stackerLoadStates.stResetDone);
  	    ELSE
			Stations.sLoadDrive.TargetPosition     := axisPosArr[currentPos];
			Stations.sLoadDrive.TargetAcceleration := Stations.sLoadSettings.axisAcc;
			Stations.sLoadDrive.TargetVelocity     := Stations.sLoadSettings.axisWorkSpeed;
			Stations.sLoadDrive.DoMove             := TRUE;
			moveDone 				    		   := FALSE;
			IF stateDelay(drivePosTime) THEN
				nextState(stackerLoadStates.stPreparePalletMoveCheck);
			END_IF
		END_IF	
		
// *** Prapare Pallet - Move Up Check
// Стакера е направил един ход нагоре
// В завизимост от това дали има тара или не се прави нов ход или се зкл. терата

	stackerLoadStates.stPreparePalletMoveCheck:
		IF Stations.sLoadDrive.TargetReached AND NOT Stations.sLoadDrive.Error THEN
			Stations.sLoadDrive.DoMove := FALSE;
			moveDone			       := TRUE;
			nextState(stackerLoadStates.stPreparePalletLock);	
		ELSIF NOT Stations.sLoadDrive.TargetReached AND Stations.sLoadDrive.Error THEN
			setError(stackerLoadStates.stErrPalletMove);
		END_IF	
		timeOutError(palletMoveTimeOut, stackerLoadStates.stErrPalletMove);
		
// *** Prapare Pallet - Lock
// В завизимост от това дали има тара или не се прави нов ход или се зкл. терата

	stackerLoadStates.stPreparePalletLock:
		IF io.getX(ioImage.xPalletOnTop) THEN
			nextState(stackerLoadStates.stPreparePalletDone);
		END_IF
		IF stateDelay(sensorTime) THEN
			IF currentPos > 0 THEN
				nextState(stackerLoadStates.stPreparePalletMove);
			ELSIF  currentPos = 0 THEN
				palletsLoadDone   := FALSE;
				nextState(stackerLoadStates.stResetDone);	
			END_IF	
		END_IF		
		
// *** Prepare Pallet - Done
// Има стигнала тара на върха на стакера
	stackerLoadStates.stPreparePalletDone:
		preparePalletDone := TRUE;
		nextState(stackerLoadStates.stMoveDownStart);

// *** Move Down - Start
// Тарата трябва да се заключи и да се направи 1 ход надолу
	stackerLoadStates.stMoveDownStart:
		moveDownDone   := FALSE;
		nextState(stackerLoadStates.stMoveDownCkeckTop);
		
// *** Move Down - Check top
// Проверява дали има тара на върха на стакера 
	stackerLoadStates.stMoveDownCkeckTop:		
		IF io.getX(ioImage.xPalletOnTop) THEN
			io.setSR(ioImage.yLocks_lock, ioImage.yLocks_unlock);
			nextState(stackerLoadStates.stMoveDownCheckLocks);
		ELSE
			preparePalletDone := FALSE;
			setError(stackerLoadStates.stErrNoPallet);
		END_IF
			
// *** Move Down - Check Locks
// Трябва всички ключалки да са затворени преди да тръгне надолу стакера

	stackerLoadStates.stMoveDownCheckLocks:
		IF io.getSR(ioImage.xLock1_lock, ioImage.xLock1_unlock) AND 
		   io.getSR(ioImage.xLock2_lock, ioImage.xLock2_unlock) THEN
		   		io.setSR(ioImage.yPalletFix_lock, ioImage.yPalletFix_unlock);
				nextState(stackerLoadStates.stMoveDownCheckFix);
		END_IF
		
		IF stateDelay(cylinderTimeOut) THEN
			
			IF NOT io.getSR(ioImage.xLock1_lock, ioImage.xLock1_unlock) THEN
				setError(stackerLoadStates.stErrLock1NotClose);
			ELSIF NOT io.getSR(ioImage.xLock2_lock, ioImage.xLock2_unlock) THEN
				setError(stackerLoadStates.stErrLock2NotClose);
				END_IF

		END_IF	
		
//  *** Move Down - Check Fix
// Проверка дали фиксиращият цилиндър е затворил

	stackerLoadStates.stMoveDownCheckFix:
		IF io.getSR(ioImage.xPalletFix_lock, ioImage.xPalletFix_unlock) THEN
			nextState(stackerLoadStates.stMoveSync);
		END_IF
		timeOutError(cylinderTimeOut,stackerLoadStates.stErrFixerNotClose);
		
//  *** Move Down - Sync

	stackerLoadStates.stMoveSync:		
		depSync(Stations.roboStBase, globalDeps.depSLoadStationReady);		
		Global.lStackerEmpty := FALSE;
		IF Stations.sLoadDrive.Enabled AND NOT Stations.sLoadDrive.Error THEN				
			nextState(stackerLoadStates.stMoveDownMove);
		ELSE
			nextState(stackerLoadStates.stMoveDownDriveOn);
		END_IF		
			
//  *** Move Down - Drive On
// Активира се мотора на оста за да направи 1 ход надолу

	stackerLoadStates.stMoveDownDriveOn:
		IF Stations.sLoadDrive.Error THEN
			Stations.sLoadDrive.DoReset  := TRUE;
		ELSE
			Stations.sLoadDrive.DoReset  := FALSE;
			Stations.sLoadDrive.DoEnable := TRUE;
			IF stateDelay(driveEnTime) AND Stations.sLoadDrive.Enabled THEN
				setDisplayState(stackerLoadDisplayStates.dStWaitForPallet);
				nextState(stackerLoadStates.stMoveDownMove);
			END_IF
		END_IF
		timeOutError(driveEnTime * 2, stackerLoadStates.stErrAxis);	
		
//  *** Move Down - Move
//  1 ход надолу
	stackerLoadStates.stMoveDownMove:
		IF moveDone THEN
			currentPos := currentPos + 1;
		END_IF
		IF currentPos >= posCount THEN
			currentPos := posCount;
		END_IF
		Stations.sLoadDrive.TargetPosition     := axisPosArr[currentPos];
		Stations.sLoadDrive.TargetAcceleration := Stations.sLoadSettings.axisAcc;
		Stations.sLoadDrive.TargetVelocity     := Stations.sLoadSettings.axisWorkSpeed;
		Stations.sLoadDrive.DoMove             := TRUE;
		moveDone						       := FALSE;
		IF stateDelay(drivePosTime) THEN
			nextState(stackerLoadStates.stMoveDownMoveCheck);
		END_IF	
		
		IF stateDelay(cylinderTimeOut) THEN
			setError(stackerLoadStates.stErrFixerNotClose);
		END_IF		
		
// *** Move Down - Move Check
// Проверка дали стакера е слезнал на поз.

	stackerLoadStates.stMoveDownMoveCheck:
		IF Stations.sLoadDrive.TargetReached AND NOT Stations.sLoadDrive.Error THEN
			Stations.sLoadDrive.DoMove := FALSE;
			moveDone			       := TRUE;
			nextState(stackerLoadStates.stMoveDownDone);	
		ELSIF NOT Stations.sLoadDrive.TargetReached AND Stations.sLoadDrive.Error THEN
			setError(stackerLoadStates.stErrPalletMove);
		END_IF	
		timeOutError(palletMoveTimeOut, stackerLoadStates.stErrPalletMove);
		
// *** Move Down - Done

	stackerLoadStates.stMoveDownDone:
		moveDownDone := TRUE;			
		nextState(stackerLoadStates.stInitDone);       // робота го ползва в stWaitLoadStacker при инициализация
		
// *** Release Pallet - Start
// Текушата тара се е изпразнила 

	stackerLoadStates.stReleasePalletStart:
		palletReleaseStart  := TRUE;
		setDisplayState(stackerLoadDisplayStates.dStReleaseEmptyPallet);
		nextState(stackerLoadStates.stReleasePalletUnlock);
	
// *** Release Pallet - Unlock
// Отключва тарата

	stackerLoadStates.stReleasePalletUnlock:	
		io.setSR(ioImage.yLocks_unlock, ioImage.yLocks_lock);
		io.setSR(ioImage.yPalletFix_unlock, ioImage.yPalletFix_lock);
		nextState(stackerLoadStates.stReleasePalletUnlockCheck);	

// *** Release Pallet - Unlock Check
// Проверка дали вички ключалки са се отворили

	stackerLoadStates.stReleasePalletUnlockCheck:	
		IF io.getSR(ioImage.xLock1_unlock, ioImage.xLock1_lock) AND 
		   io.getSR(ioImage.xLock2_unlock, ioImage.xLock2_lock) AND
		   io.getSR(ioImage.xPalletFix_unlock, ioImage.xPalletFix_lock) THEN
		   		nextState(stackerLoadStates.stReleasePalletSignalRobot);
		END_IF
		
		IF stateDelay(cylinderTimeOut) THEN
			
			IF NOT io.getSR(ioImage.xLock1_unlock, ioImage.xLock1_lock) THEN
				setError(stackerLoadStates.stErrLock1NotOpen);
			ELSIF NOT io.getSR(ioImage.xLock2_unlock, ioImage.xLock2_lock) THEN
				setError(stackerLoadStates.stErrLock2NotOpen);
			ELSIF NOT io.getSR(ioImage.xPalletFix_unlock, ioImage.xPalletFix_lock) THEN
				setError(stackerLoadStates.stErrFixerNotOpen);
		    END_IF
		END_IF
		
// *** Release Pallet - Signal Robot
// Тарата е свободна и робота може да я мести

	stackerLoadStates.stReleasePalletSignalRobot:	
		depSync(Stations.roboStBase, GlobalDeps.depRoboLoadPalletUnlock);	
		nextState(stackerLoadStates.stReleasePalletDone);	
		
// *** Release Pallet - Done

	stackerLoadStates.stReleasePalletDone:
		palletReleaseStart  := FALSE;	
		nextState(stackerLoadStates.stRoboOutStart);
		
// ***  Robot Out - Start
// Изчаква робота да се премести на безопастно разтояние

	stackerLoadStates.stRoboOutStart:	
		roboOutStart := TRUE;
		depNextState(Stations.roboStBase, globalDeps.depRoboStartLoadStacker, stackerLoadStates.stRoboOutDone);
		
// ***  Robot Out - Done

	stackerLoadStates.stRoboOutDone:	
		roboOutStart := FALSE;	
		nextState(stackerLoadStates.stInitDone);	
		
// *** Purge - Start
// Без значение колко палети има те трябва да се извадят от стакера

	stackerLoadStates.stLoadPurgeStart:
		purgeStart  := TRUE;
		setDisplayState(stackerLoadDisplayStates.dStStackerIsReseting);  // Purge си е просто втори вид Reset
		nextState(stackerLoadStates.stLoadPurgeCheck);
		
// *** Purge - Check
// Ако стакера е на горна крайна поз. - се прави Reset

	stackerLoadStates.stLoadPurgeCheck:
		IF moveDone AND currentPos = 0 THEN
			nextState(stackerLoadStates.stLoadPurgeDone);
		ELSE
			IF Stations.sLoadDrive.Enabled AND NOT Stations.sLoadDrive.Error THEN
				nextState(stackerLoadStates.stLoadPurgeMove);
			 ELSE
				nextState(stackerLoadStates.stLoadPurgeDriveOn);
			END_IF	
		END_IF
		
//  *** Purge - Drive On 
// Проверява дали всичко е наред с мотора

	stackerLoadStates.stLoadPurgeDriveOn:
		IF Stations.sLoadDrive.Error THEN
			Stations.sLoadDrive.DoReset  := TRUE;
		ELSE
			Stations.sLoadDrive.DoReset  := FALSE;
			Stations.sLoadDrive.DoEnable := TRUE;
			IF stateDelay(driveEnTime) THEN
				nextState(stackerLoadStates.stLoadPurgeMove);
			END_IF
		END_IF
		timeOutError(driveEnTime * 2, stackerLoadStates.stErrAxis);	

// *** Purge- Move
// Прества стакера нагоре с 1 поз. нагоре

	stackerLoadStates.stLoadPurgeMove:
		IF moveDone THEN
			currentPos := currentPos - 1;
		END_IF
		IF currentPos <= 0 THEN
			currentPos := 0; 
		END_IF
		Stations.sLoadDrive.TargetPosition     := axisPosArr[currentPos];
		Stations.sLoadDrive.TargetAcceleration := Stations.sLoadSettings.axisAcc;
		Stations.sLoadDrive.TargetVelocity     := Stations.sLoadSettings.axisWorkSpeed;
		Stations.sLoadDrive.DoMove             := TRUE;
		moveDone 				    		   := FALSE;
		IF stateDelay(drivePosTime) THEN
			nextState(stackerLoadStates.stLoadPurgeMoveCheck);
        END_IF	
		
// *** Purge - Move Check
// Стакера е направил един ход нагоре

	stackerLoadStates.stLoadPurgeMoveCheck:
		IF Stations.sLoadDrive.TargetReached AND NOT Stations.sLoadDrive.Error THEN
			Stations.sLoadDrive.DoMove := FALSE;
			moveDone			       := TRUE;
			nextState(stackerLoadStates.stLoadPurgeDone);	
		ELSIF NOT Stations.sLoadDrive.TargetReached AND Stations.sLoadDrive.Error THEN
			setError(stackerLoadStates.stErrPalletMove);
		END_IF	
		timeOutError(palletMoveTimeOut, stackerLoadStates.stErrPalletMove);	

// *** Purge - Done
// От тук стакера се ресетва

	stackerLoadStates.stLoadPurgeDone:	
		nextState(stackerLoadStates.stResetStart);
	
// *** Step Block State
// В този state се влиза винаги след изпълняването на една стъпка при стъпков режим
	stackerLoadStates.stStepBlock:
		setDisplayState(stackerLoadDisplayStates.dStWaitForNextStep);
		
// *** Station Stop
// Станцията е била изключена 
 
	stackerLoadStates.stStop: 						   							   
		resetDone			          := FALSE; 						   
		palletsLoadDone		          := FALSE;							   
		preparePalletDone             := FALSE; 						   
		palletReleaseStart	          := FALSE; 
		moveDownDone			      := FALSE;	
	    purgeStart					  := FALSE;					  
		moveDone		              := FALSE; 
		Stations.sLoadDrive.DoMove    := FALSE;
		Stations.sLoadDrive.DoEnable  := FALSE;	
		setDisplayState(stackerLoadDisplayStates.dStStationIsStopped);
	
// Състояния за грешки
	
//  *** ERROR No axis setting
// 	Липсват настойки на оста (ход и размер на тара)	

	stackerLoadStates.stErrNoProperSettings:
		setDisplayState(stackerLoadDisplayStates.dStAxisNotConfigured);

// *** ERROR remove Pallet	
// След старт на машината не трябва да има палет на стакера. 
// Ако има оператора трябва да го махне

	stackerLoadStates.stErrRemovePallet:
		setDisplayState(stackerLoadDisplayStates.dStRemotePalletManually);

// *** ЕRROR  Lock 1 not open
// Цилиндъра не се е отворил навреме
		
	stackerLoadStates.stErrLock1NotOpen:
		setDisplayState(stackerLoadDisplayStates.dStLock1CylinderDidNotOpen);
		
// *** ЕRROR  Lock 1 not close
// Цилиндъра не се е затворил навреме
		
	stackerLoadStates.stErrLock1NotClose:
		setDisplayState(stackerLoadDisplayStates.dStLock1CylinderDidNotClose);	
		
// *** ЕRROR  Lock 2 not open
// Цилиндъра не се е отворил навреме	
	
	stackerLoadStates.stErrLock2NotOpen:
		setDisplayState(stackerLoadDisplayStates.dStLock2CylinderDidNotOpen);		
		
// *** ЕRROR  Lock 2 not close
// Цилиндъра не се е затворил навреме	
	
	stackerLoadStates.stErrLock2NotClose:
		setDisplayState(stackerLoadDisplayStates.dStLock2CylinderDidNotClose);			

// *** ЕRROR  Fixer not open
// Цилиндъра не се е отворил навреме	
	
	stackerLoadStates.stErrFixerNotOpen:
		setDisplayState(stackerLoadDisplayStates.dStFixerCylinderDidNotOpen);	
		
// *** ЕRROR  Fixer not close
// Цилиндъра не се е затворил навреме	
	
	stackerLoadStates.stErrFixerNotClose:
		setDisplayState(stackerLoadDisplayStates.dStFixerCylinderDidNotClose);		

// *** ERROR Axis
// Има грешка на FESTO инвертора

	stackerLoadStates.stErrAxis:
		Stations.sLoadDrive.DoEnable     := FALSE;
		setDisplayState(stackerLoadDisplayStates.dStFestoDriveError);
		
// ***ERROR Init move
// Движението към горна крайна точка при init е отнело твърде мн. време		
		
	stackerLoadStates.stInitMoveErr:
		Stations.sLoadDrive.DoMove       := FALSE;
		Stations.sLoadDrive.DoEnable     := FALSE;
		setDisplayState(stackerLoadDisplayStates.dStAxisInitMoveTakesTooLong);
		
// *** ERROR Pallet Load 
// Движението при зареждане на тарите е отнело твърде мн време

	stackerLoadStates.stErrPalletLoad:
		Stations.sLoadDrive.DoMove       := FALSE;
		Stations.sLoadDrive.DoEnable     := FALSE;
		setDisplayState(stackerLoadDisplayStates.dStPalletLoadMoveTakesTooLong);
		
// *** ERROR Pallet Move up
// Движението за преместването на една тара ход нагоре е отнело твърде мн време

	stackerLoadStates.stErrPalletMove:
		Stations.sLoadDrive.DoMove       := FALSE;
		Stations.sLoadDrive.DoEnable     := FALSE;
		setDisplayState(stackerLoadDisplayStates.dStPalletMoveTakesTooLong);

// *** ERROR No Pallet
// Стакер се опитва да зареди тари, но не открива тара на върха

	stackerLoadStates.stErrNoPallet:
		setDisplayState(stackerLoadDisplayStates.dStThereIsNoPalletOnTop);		
		
// *** EMG Stop
// Аварийно спиране при натискане на гъба или отваряне на врата

	stackerLoadStates.stEMG:	
		
		Stations.sLoadDrive.DoMove       := FALSE;
		Stations.sLoadDrive.DoEnable     := FALSE;
		
		nextState(stackerLoadStates.stInit);
	
END_CASE

ACTION drivesControl:


axisFesto          ( axis				:= Stations.sLoadAxis,
					PowerUP 			:= Stations.sLoadDrive.DoEnable, 
					Home 				:= Stations.sLoadDrive.DoHome, 
					StartMove 			:= Stations.sLoadDrive.DoMove, 
					Reset 				:= Stations.sLoadDrive.DoReset, 
					Position 			:= Stations.sLoadDrive.TargetPosition, 
					Velocity 			:= Stations.sLoadDrive.TargetVelocity,
					Acceleration		:= Stations.sLoadDrive.TargetAcceleration,
					IsAbsolute 			:= TRUE,
					Enabled 			=> Stations.sLoadDrive.Enabled,
					Error 				=> Stations.sLoadDrive.Error,
					ErrorID 			=> Stations.sLoadDrive.ErrorID,
					TargetReached 		=> Stations.sLoadDrive.TargetReached,
					HomeDone 			=> Stations.sLoadDrive.Refferenced,
					Moving 				=> Stations.sLoadDrive.Moving,
					CurrentPosition 	=> Stations.sLoadDrive.CurrentPosition,
					OperationMode		=> Stations.sLoadDrive.OperationMode);
END_ACTION

END_FUNCTION_BLOCK

// ---- POUs/Stations/stackerUnloadStation.TcPOU
FUNCTION_BLOCK stackerUnloadStation EXTENDS stateMachine
VAR_INPUT
	
	ioImage                : stackerUnloadImage;

END_VAR

VAR

	activeState            : stackerUnloadStates;	
	axisFesto              : FB_FESTO_CMMT_AS;
	

	resetDone			   : BOOL := FALSE; 						   //  След подава не захр. станцията се е ресетната
	prepareDone			   : BOOL := FALSE;							   //  Стакера е на позиция - станцията е готова за работа
	moveUpStart			   : BOOL := FALSE;							   //  Стакера се е преместил точно под тарата
	unlockPalletStart      : BOOL := FALSE; 						   //  Тарата е оключена и е на стакера - може да се премести надолу
	fixPalletStart		   : BOOL := FALSE; 						   //  Робота е доставил нова тара - може да се фиксира
	purgeStart			   : BOOL := FALSE; 						   //  Purge на станцията е завършил	
	
	moveDone		       : BOOL := FALSE; 						   // Фесто мотора си е изпълнил заданието при движение
	moveInit			   : BOOL;
	
	posCount			   : DINT;					 				   // Брой позиций на оста
	axisLen				   : REAL;				
	currentPos 			   : DINT;					 				   // Текуща позиция
	axisPosArr			   : ARRAY [0..Consts.MAX_AXIS_POS] OF REAL;   // Масив с позицийте на оста
	
	cylinderTimeOut		   : TIME := T#2S;                             // Време за ход на цилиндър
	driveEnTime		       : TIME := T#1S;							   // Време за enable на фесто drive
	initMoveTimeOut		   : TIME := T#20S;                            // Време за ход до крайно горно положение
	sensorTime 			   : TIME := T#250MS;                          // Време за реакция на оптичен сензор
	palletsLoadTimeOut	   : TIME := T#15S; 						   // Време за ход на зареждане на тари
	palletMoveTimeOut	   : TIME := T#10S;                            // Време за преместване на 1 позиция
	drivePosTime           : TIME := T#100MS;                          // Време за задаване на задание за позициониране



END_VAR


drivesControl();          // Упр. на Феесто мотора дрижещ осна на стакера

setStateVars(ioImage, activeState);


CASE activeState OF 
	
//  *** Start Up
//  Старт на станцията след подаване на захр.	

	stackerUnloadStates.stStartUp:
		setDisplayState(stackerUnLoadDisplayStates.dStStartingUp);
		Stations.sUnloadDrive.DoEnable  := FALSE;
		Stations.sUnloadDrive.DoMove    := FALSE;						   						   
		nextState(stackerUnloadStates.stPowerUp);
		
//  *** Power Up - Start
//  Инициализация след подaване на захранване

	stackerUnloadStates.stPowerUp:
		IF io.getX(ioImage.xPalletOnTop) THEN
			setError(stackerUnloadStates.stErrRemovePallet);
		END_IF
		
//  *** Init 
//  Инициализация на станцията
	
	stackerUnloadStates.stInit:
	
		depWait(globalDeps.depSUnloadInit);		

		// Проверка за приключила инициализация - стакера е горе, празен
		IF NOT resetDone THEN
			nextState(stackerUnloadStates.stResetStart);
	    END_IF	
		
		// Стакера е  на позиция за работа - 1 ход под върха си
		IF NOT prepareDone THEN
			nextState(stackerUnloadStates.stPrepareStart);		
		END_IF
		
		// Стакера е в горна крайна позиция
		IF moveUpStart THEN
			nextState(stackerUnloadStates.stMoveUpStart);		
		END_IF
		
		// Има освободена тара на върха на стакера - може да се заради
		IF unlockPalletStart  THEN
			nextState(stackerUnloadStates.stUnlockPalletStart);
		END_IF
		
		// Стакера е заключил тара доставена от робота
		IF fixPalletStart  THEN
			nextState(stackerUnloadStates.stLockPalletLockFix);
		END_IF		
		
		// Проверява дали е приключила PURGE  процедура
		IF purgeStart THEN
			nextState(stackerUnloadStates.stUnloadPurgeStart);
		END_IF
		
		nextState(stackerUnloadStates.stInitDone);
		
// *** Init Done
// След излизането от аварийна ситуация или след изчисването на грешка
// станция е завършила своята инициализация

	stackerUnloadStates.stInitDone:

		nextState(stackerUnloadStates.stReady);	
		
// *** Ready

	stackerUnloadStates.stReady:
		setDisplayState(stackerUnLoadDisplayStates.dStStandBy);
		depNextState(Stations.machineStBase,  globalDeps.depMachineStopping,      stackerUnloadStates.stStackerStopped);
		depNextState(Stations.machineStBase,  globalDeps.depMachineStop,          stackerUnloadStates.stStackerStopped);		
		depNextState(Stations.roboStBase,     globalDeps.depRoboUnLodPalletFull,  stackerUnloadStates.stMoveUpStart);
	    depNextState(Stations.machineStBase,  globalDeps.depMacinePurgeStackers,  stackerUnloadStates.stUnloadPurgeStart);		
		depWait(globalDeps.depSUnloadRobotUnloadGrip);
		nextState(stackerUnloadStates.stLockPalletStart);
		
// *** Stacker is Stopped
// Стакера е спрял след като е завършил текущият си цикъл и е бил натиснат STOP бутона

	stackerUnloadStates.stStackerStopped:
        setDisplayState(stackerUnLoadDisplayStates.dStStationIsStopped);	
		Stations.sUnloadDrive.DoMove       := FALSE;
		Stations.sUnloadDrive.DoEnable     := FALSE;
		depWait(GlobalDeps.depSUnloadStop);	
		depNextState(stations.machineStBase, globalDeps.depMachineAuto,       stackerUnloadStates.stInitDone);
		depNextState(stations.machineStBase, globalDeps.depMachinePurgeStart, stackerUnloadStates.stReady);

// *** Reset - Start
// Започва инициялизация на стакера - трябва да се премести 
// нагоре докрай. Затова първо робота трябва да е на безопасно място.	

	stackerUnloadStates.stResetStart:
		resetDone   := FALSE;
		setDisplayState(stackerUnLoadDisplayStates.dStStackerIsReseting);
		IF NOT Global.robotSafe THEN
			depWait(globalDeps.depSUnloadWaitRobotReady);
			nextState(stackerUnloadStates.stResetOpenLocks);
		ELSE
			nextState(stackerUnloadStates.stResetOpenLocks);				
		END_IF
		
// *** Reset - Open Locks
// Отваряне на всички ключалки	

	stackerUnloadStates.stResetOpenLocks:
		io.setSR(ioImage.yLocks_unlock, ioImage.yLocks_lock);
		io.setSR(ioImage.yPalletFix_unlock, ioImage.yPalletFix_lock);
		nextState(stackerUnloadStates.stResetCheckLocks);

// *** Reset - Check Locks
// Проверка дали всички ключалки са отворени	

	stackerUnloadStates.stResetCheckLocks:	   
		IF io.getSR(ioImage.xLock1_unlock, ioImage.xLock1_lock) AND 
		   io.getSR(ioImage.xLock2_unlock, ioImage.xLock2_lock) AND
		   io.getSR(ioImage.xPalletFix_unlock, ioImage.xPalletFix_lock) THEN
		   		nextState(stackerUnloadStates.stResetEnableDrive);
		END_IF
		
		IF stateDelay(cylinderTimeOut) THEN
			
			IF NOT io.getSR(ioImage.xLock1_unlock, ioImage.xLock1_lock) THEN
				setError(stackerUnloadStates.stErrLock1NotOpen);
			ELSIF NOT io.getSR(ioImage.xLock2_unlock, ioImage.xLock2_lock) THEN
				setError(stackerUnloadStates.stErrLock2NotOpen);
			ELSIF NOT io.getSR(ioImage.xPalletFix_unlock, ioImage.xPalletFix_lock) THEN
				setError(stackerUnloadStates.stErrFixerNotOpen);
		    END_IF
			
		END_IF 
		
// *** Reset - Enable Drive
// Вкл. на инвертора на FESTO мотора на оста на стакера	

	stackerUnloadStates.stResetEnableDrive:
		IF Stations.sUnloadDrive.Error THEN
			Stations.sUnloadDrive.DoReset  := TRUE;
		ELSE
			Stations.sUnloadDrive.DoReset  := FALSE;
			Stations.sUnloadDrive.DoEnable := TRUE;
			IF stateDelay(driveEnTime) THEN
				nextState(stackerUnloadStates.stResetDriveMove);
			END_IF
		END_IF
		timeOutError(driveEnTime*2, stackerUnLoadStates.stErrAxis);

// *** Reset - Drive Move
// Оста на стакера прави ход до горно крайно положение

	stackerUnloadStates.stResetDriveMove:	
		IF Stations.sUnloadDrive.Enabled AND NOT Stations.sUnloadDrive.Error THEN
			Stations.sUnloadDrive.TargetPosition     := Stations.sUnloadSettings.pallet[Global.recipe].zeroPos;
			Stations.sUnloadDrive.TargetAcceleration := Stations.sUnloadSettings.axisAcc;
			Stations.sUnloadDrive.TargetVelocity     := Stations.sUnloadSettings.axisInitSpeed;
			Stations.sUnloadDrive.DoMove             := TRUE;
			moveDone							     := FALSE;
			IF stateDelay(drivePosTime) THEN
				nextState(stackerUnloadStates.stResetCheckDrive);
			END_IF
		ELSE
			setError(stackerUnloadStates.stErrAxis);
	   END_IF	

// *** Reset - Check Drive
// Проверка дали оста е завършила хода си - горно крайно положение

	stackerUnloadStates.stResetCheckDrive:	
		IF Stations.sUnloadDrive.TargetReached AND NOT Stations.sUnloadDrive.Error THEN
			Stations.sUnloadDrive.DoMove := FALSE;
			moveDone 				     := TRUE;
			nextState(stackerUnloadStates.stResetDone);	
		ELSIF NOT Stations.sUnloadDrive.TargetReached AND Stations.sUnloadDrive.Error THEN
			setError(stackerUnloadStates.stInitMoveErr);
		END_IF	
		timeOutError(initMoveTimeOut, stackerUnloadStates.stInitMoveErr);			

// *** Reset - Done

	stackerUnloadStates.stResetDone:
		IF NOT purgeStart THEN		
			resetDone   			    := TRUE;
			prepareDone 			    := FALSE;
			tagsHMI.UnloadStackerSignal := TRUE;
		ELSE
			nextState(stackerUnloadStates.stUnloadPurgeConfirm);
		END_IF	

// *** Purge - Confirm
// Този state се изпълнява само при край на PURGE - за може правилно да завърши тази процедура

	stackerUnloadStates.stUnloadPurgeConfirm:
		 purgeStart                  := FALSE;	
		 resetDone                   := TRUE;		
		 prepareDone                 := FALSE;
		 tagsHMI.UnloadStackerSignal := TRUE;
		 depWait(globalDeps.depSUnloadPurgeDone);
				
// *** Prepare - Start
// Стакера трябва да стой на 1 ход под горна крайна точка

	stackerUnloadStates.stPrepareStart:
		prepareDone := FALSE;
		nextState(stackerUnloadStates.stPreparaCheckTop);
				
// *** Prepare - Check Top
// На върха на стакера не трябва да има тари 

	stackerUnloadStates.stPreparaCheckTop:		
		IF NOT io.getX(ioImage.xPalletOnTop) THEN
			nextState(stackerUnloadStates.stPrepareLimitCheck);
		ELSE
			setError(stackerUnloadStates.stErrPalletDetected);
		END_IF
		
// *** Prepare - Limit Check
//  Проверяват се дали има зададени параметри на хода на стакера
//  Ако няма такива НЕ може да се продължи с инизиализацията

	stackerUnloadStates.stPrepareLimitCheck:
		IF Stations.sUnloadSettings.axisLength < Consts.MIN_AXIS_LEN OR Stations.sUnloadSettings.pallet[Global.recipe].moveDownStep < Consts.MIN_PALLET_SIZE THEN
				setError(stackerUnloadStates.stErrNoProperSettings);
		END_IF
		nextState(stackerUnloadStates.stPrepareCalcAxis);			

// *** Prepare - Calc Axis
// Изчисляват се позицийте за хода на оста на стакера 	

	stackerUnloadStates.stPrepareCalcAxis:
	    axisLen       := Stations.sUnloadSettings.pallet[Global.recipe].zeroPos;
		axisPosArr[0] := Stations.sUnloadSettings.pallet[Global.recipe].zeroPos;
		currentPos 	  := 1;
		posCount      := 1;
		
		WHILE axisLen < Stations.sUnloadSettings.axisLength AND currentPos < Consts.MAX_AXIS_POS DO
			axisLen    			   := axisLen + Stations.sUnloadSettings.pallet[Global.recipe].moveDownStep;
			axisPosArr[currentPos] := axisLen;
			currentPos  := currentPos + 1;
			axisLen    			   := axisLen - Stations.sUnloadSettings.pallet[Global.recipe].moveUpStep;
			axisPosArr[currentPos] := axisLen;
			currentPos  := currentPos + 1;
		END_WHILE
		
		posCount     := currentPos;
		currentPos   := 0;
		nextState(stackerUnloadStates.stPrepareOpenLocks);

// *** Prepare - Open Lock
// Отваряне на всички ключалки	

	stackerUnloadStates.stPrepareOpenLocks:		
		io.setSR(ioImage.yLocks_unlock, ioImage.yLocks_lock);
		io.setSR(ioImage.yPalletFix_unlock, ioImage.yPalletFix_lock);
		nextState(stackerUnloadStates.stPrepareCheckLocks);	

// *** Prepare - Check Locks
// Проверка дали всички ключалки са отворени	

	stackerUnloadStates.stPrepareCheckLocks:	   
		IF io.getSR(ioImage.xLock1_unlock, ioImage.xLock1_lock) AND 
		   io.getSR(ioImage.xLock2_unlock, ioImage.xLock2_lock) AND
		   io.getSR(ioImage.xPalletFix_unlock, ioImage.xPalletFix_lock) THEN
		   		nextState(stackerUnloadStates.stPrepareDriveOn);
		END_IF
		
		IF stateDelay(cylinderTimeOut) THEN
			
			IF NOT io.getSR(ioImage.xLock1_unlock, ioImage.xLock1_lock) THEN
				setError(stackerUnloadStates.stErrLock1NotOpen);
			ELSIF NOT io.getSR(ioImage.xLock2_unlock, ioImage.xLock2_lock) THEN
				setError(stackerUnloadStates.stErrLock2NotOpen);
			ELSIF NOT io.getSR(ioImage.xPalletFix_unlock, ioImage.xPalletFix_lock) THEN
				setError(stackerUnloadStates.stErrFixerNotOpen);
		    END_IF
			
		END_IF	

// *** Prepare - Drive On
// Изчисляват се позицийте за хода на оста на стакера 	

	stackerUnloadStates.stPrepareDriveOn:
		IF Stations.sUnloadDrive.Error THEN
			Stations.sUnloadDrive.DoReset  := TRUE;
		ELSE
			Stations.sUnloadDrive.DoReset  := FALSE;
			Stations.sUnloadDrive.DoEnable := TRUE;
			IF stateDelay(driveEnTime) THEN
				nextState(stackerUnloadStates.stPrepareDriveMove);
			END_IF
		END_IF
		timeOutError(driveEnTime*2, stackerUnloadStates.stErrAxis);
	
		
// *** Prepare - Drive Move
// Оста на стакера прави ход 1 поз. под крайната горна точка

	stackerUnloadStates.stPrepareDriveMove:	
		IF Stations.sUnloadDrive.Enabled AND NOT Stations.sUnloadDrive.Error THEN
			currentPos								 := 1;
			Stations.sUnloadDrive.TargetPosition     := axisPosArr[currentPos];
			Stations.sUnloadDrive.TargetAcceleration := Stations.sUnloadSettings.axisAcc;
			Stations.sUnloadDrive.TargetVelocity     := Stations.sUnloadSettings.axisInitSpeed;
			Stations.sUnloadDrive.DoMove             := TRUE;
			moveDone							     := FALSE;
			moveInit								 := FALSE;
			IF stateDelay(drivePosTime) THEN
				nextState(stackerUnloadStates.stPrepareCheckDrive);
			END_IF
		ELSE
			setError(stackerUnloadStates.stErrAxis);
	   END_IF			
	
// *** Prepare - Check Drive
// Проверка дали оста е завършила хода си - 1 поз. под горна крайна точка

	stackerUnloadStates.stPrepareCheckDrive:		
		IF Stations.sUnloadDrive.TargetReached AND NOT Stations.sUnloadDrive.Error THEN
			Stations.sUnloadDrive.DoMove := FALSE;
			moveDone 				     := TRUE;
			nextState(stackerUnloadStates.stPrepareSync);	
		ELSIF NOT Stations.sUnloadDrive.TargetReached AND Stations.sUnloadDrive.Error THEN
			setError(stackerUnloadStates.stInitMoveErr);
		END_IF	
		timeOutError(palletMoveTimeOut, stackerUnloadStates.stErrPalletMove);	
		
// *** Prepare - Sync

	stackerUnloadStates.stPrepareSync:		
		depWait(globalDeps.depSUnloadStationReady);	
		nextState(stackerUnloadStates.stPrepareDone);			
		
// *** Prepare - Done

	stackerUnloadStates.stPrepareDone:		
		prepareDone         := TRUE;
		Global.uStackerFull := FALSE;
		nextState(stackerUnloadStates.stReady);		
	
// *** Move up - Start
// Прави се 1 ход нагоре  - стакера застава под тарата

	stackerUnloadStates.stMoveUpStart:	
		moveUpStart := TRUE;
		setDisplayState(stackerUnLoadDisplayStates.dStPalletReady);
		IF Stations.sUnloadDrive.Enabled AND NOT Stations.sUnloadDrive.Error THEN
			nextState(stackerUnloadStates.stMoveUpDriveMove);
		ELSE
			nextState(stackerUnloadStates.stMoveUpDriveOn);
	    END_IF
		
// *** Move up - Drive On
// Вкл. на инвертора на FESTO мотора на оста на стакера	

	stackerUnloadStates.stMoveUpDriveOn:	
		IF Stations.sUnloadDrive.Error THEN
			Stations.sUnloadDrive.DoReset  := TRUE;
		ELSE
			Stations.sUnloadDrive.DoReset  := FALSE;
			Stations.sUnloadDrive.DoEnable := TRUE;
			IF stateDelay(driveEnTime) THEN
				nextState(stackerUnloadStates.stMoveUpDriveMove);
			END_IF
		END_IF
		timeOutError(driveEnTime*2, stackerUnloadStates.stErrAxis);
	
// *** Move up - Drive Move
// Прави 1 ход нагоре

	stackerUnloadStates.stMoveUpDriveMove:	
		IF moveDone AND moveInit THEN
			currentPos := currentPos + 1;
		ELSIF moveDone AND NOT moveInit THEN
			currentPos := 0;
		END_IF
		Stations.sUnloadDrive.TargetPosition     := axisPosArr[currentPos];
		Stations.sUnloadDrive.TargetAcceleration := Stations.sUnloadSettings.axisAcc;
		Stations.sUnloadDrive.TargetVelocity     := Stations.sUnloadSettings.axisInitSpeed;
		Stations.sUnloadDrive.DoMove             := TRUE;
		moveDone							     := FALSE;
		IF stateDelay(drivePosTime) THEN		
			nextState(stackerUnloadStates.stMoveUpCkeckDrive);
		END_IF	
	
// *** Move up - Check Drive
// Проверка дали е завършил хода на оста

	stackerUnloadStates.stMoveUpCkeckDrive:		
		IF Stations.sUnloadDrive.TargetReached AND NOT Stations.sUnloadDrive.Error THEN
			Stations.sUnloadDrive.DoMove := FALSE;
			moveDone 				     := TRUE;
			nextState(stackerUnloadStates.stMoveUpDone);	
		ELSIF NOT Stations.sUnloadDrive.TargetReached AND Stations.sUnloadDrive.Error THEN
			setError(stackerUnloadStates.stInitMoveErr);
		END_IF	
		timeOutError(palletMoveTimeOut, stackerUnloadStates.stErrPalletMove);	
	
// *** Move up - Done

	stackerUnloadStates.stMoveUpDone:	
		moveUpStart := FALSE;	
		nextState(stackerUnloadStates.stUnlockPalletStart);
		
// *** Unlock Pallet - Start
// Освобождава пале на върха на стакера

	stackerUnloadStates.stUnlockPalletStart:	
		unlockPalletStart := TRUE;		
		nextState(stackerUnloadStates.stUnlockPalletRelease);			
		
// *** Unlock Pallet - Start
// Освобождаване на палето

	stackerUnloadStates.stUnlockPalletRelease:			
		io.setSR(ioImage.yLocks_unlock, ioImage.yLocks_lock);
		io.setSR(ioImage.yPalletFix_unlock, ioImage.yPalletFix_lock);
		nextState(stackerUnloadStates.stUnlockPalletCheck);		
	
// *** Unlock Pallet - Check
// Проверка дали са се отворили всички ключалки

	stackerUnloadStates.stUnlockPalletCheck:		
		IF io.getSR(ioImage.xLock1_unlock, ioImage.xLock1_lock) AND 
		   io.getSR(ioImage.xLock2_unlock, ioImage.xLock2_lock) AND
		   io.getSR(ioImage.xPalletFix_unlock, ioImage.xPalletFix_lock) THEN
				IF Stations.sUnloadDrive.Enabled AND NOT Stations.sUnloadDrive.Error THEN
					nextState(stackerUnloadStates.stUnlockPalletDriveMove);
				ELSE
					nextState(stackerUnloadStates.stUnlockPalletDriveOn);
	    		END_IF
		END_IF
		
		IF stateDelay(cylinderTimeOut) THEN
			
			IF NOT io.getSR(ioImage.xLock1_unlock, ioImage.xLock1_lock) THEN
				setError(stackerUnloadStates.stErrLock1NotOpen);
			ELSIF NOT io.getSR(ioImage.xLock2_unlock, ioImage.xLock2_lock) THEN
				setError(stackerUnloadStates.stErrLock2NotOpen);
			ELSIF NOT io.getSR(ioImage.xPalletFix_unlock, ioImage.xPalletFix_lock) THEN
				setError(stackerUnloadStates.stErrFixerNotOpen);
		    END_IF
			
		END_IF		
	
// *** Unlock Pallet - Drive On
// Вкл. на инвертора на FESTO мотора на оста на стакера	

	stackerUnloadStates.stUnlockPalletDriveOn:	
		IF Stations.sUnloadDrive.Error THEN
			Stations.sUnloadDrive.DoReset  := TRUE;
		ELSE
			Stations.sUnloadDrive.DoReset  := FALSE;
			Stations.sUnloadDrive.DoEnable := TRUE;
			IF stateDelay(driveEnTime) THEN
				nextState(stackerUnloadStates.stUnlockPalletDriveMove);
			END_IF
		END_IF
		timeOutError(driveEnTime*2, stackerUnloadStates.stErrAxis);	
		
// *** Unlock Pallet - Drive Move
// Прави ход надолу

	stackerUnloadStates.stUnlockPalletDriveMove:	
		IF currentPos = posCount THEN                         // Стакера е пълен
			unlockPalletStart   := FALSE;
			Global.startZumer   := TRUE;
			Global.uStackerFull := TRUE;
			nextState(stackerUnloadStates.stResetOpenLocks);
		ELSE
			IF moveDone AND moveInit THEN
				currentPos := currentPos + 1;
			ELSIF moveDone AND NOT moveInit THEN
				currentPos :=  1;	
			    moveInit   := TRUE;
			END_IF		
			IF currentPos >= posCount THEN
				currentPos := posCount;
			END_IF
			Stations.sUnloadDrive.TargetPosition     := axisPosArr[currentPos];
			Stations.sUnloadDrive.TargetAcceleration := Stations.sUnloadSettings.axisAcc;
			Stations.sUnloadDrive.TargetVelocity     := Stations.sUnloadSettings.axisInitSpeed;
			Stations.sUnloadDrive.DoMove             := TRUE;
			moveDone							     := FALSE;
		    nextState(stackerUnloadStates.stUnlockPalletCkeckDrive);
	   END_IF	
		
// *** Unlock Pallet - Check Drive
// Проверка дали е завършил хода на оста

	stackerUnloadStates.stUnlockPalletCkeckDrive:	
		IF stateDelay(drivePosTime) THEN
			IF Stations.sUnloadDrive.TargetReached AND NOT Stations.sUnloadDrive.Error THEN
				Stations.sUnloadDrive.DoMove := FALSE;
				moveDone 				     := TRUE;
				nextState(stackerUnloadStates.stUnlockPalletSync);	
			ELSIF NOT Stations.sUnloadDrive.TargetReached AND Stations.sUnloadDrive.Error THEN
				setError(stackerUnloadStates.stInitMoveErr);
			END_IF	
		END_IF	
		timeOutError(palletMoveTimeOut, stackerUnloadStates.stErrPalletMove);

// *** Unlock Pallet - Sync

	stackerUnloadStates.stUnlockPalletSync:	
		depWait(globalDeps.depSUnloadStationReady);	 
		nextState(stackerUnloadStates.stUnlockPalletDone);
		
// *** Unlock Pallet - Done

	stackerUnloadStates.stUnlockPalletDone:	
		unlockPalletStart := FALSE;
		nextState(stackerUnloadStates.stReady);	
	
// *** Lock Pallet - Start
// Робота е преместил нова тара на върха на стакера - тя трябва да се заключи

	stackerUnloadStates.stLockPalletStart:	
		setDisplayState(stackerUnLoadDisplayStates.dStStartingUp);		
		nextState(stackerUnloadStates.stLockPalletLocking);

// *** Lock Pallet - Locking
// Затваряне на ключалките, само ако има тара

	stackerUnloadStates.stLockPalletLocking: 
	IF io.getX(ioImage.xPalletOnTop) THEN
		io.setSR(ioImage.yLocks_lock, ioImage.yLocks_unlock);		
		nextState(stackerUnloadStates.stLockPalletCheckLocks);		
	END_IF
	IF stateDelay(sensorTime) THEN 
		Global.palletFail := TRUE;
		setError(stackerUnloadStates.stErrNoPallet);
	END_IF
		
// *** Lock Pallet - Check Locks
// Проверка дали ключалките са заключени

	stackerUnloadStates.stLockPalletCheckLocks:			
		IF io.getSR(ioImage.xLock1_lock, ioImage.xLock1_unlock) AND 
		   io.getSR(ioImage.xLock2_lock, ioImage.xLock2_unlock) THEN
		   		nextState(stackerUnloadStates.stLockPalletSyncRobot);
		END_IF
		
		IF stateDelay(cylinderTimeOut) THEN
			
			IF NOT io.getSR(ioImage.xLock1_lock, ioImage.xLock1_unlock) THEN
				setError(stackerUnloadStates.stErrLock1NotClose);
			ELSIF NOT io.getSR(ioImage.xLock2_lock, ioImage.xLock2_unlock) THEN
				setError(stackerUnloadStates.stErrLock2NotClose);
			END_IF
			
		END_IF		
		
// *** Lock Pallet - Synck Robot
// Тарата е заключена - робота може да освободи

	stackerUnloadStates.stLockPalletSyncRobot:			
		depSync(Stations.roboStBase, globalDeps.depRoboUnLoadPalletLock);		
		depWait(globalDeps.depSUnloadRobotOutOfReach);
		nextState(stackerUnloadStates.stLockPalletLockFix);	

// *** Lock Pallet - Lock Fix
// Робота е освободил тарата - тя може да се фиксира

	stackerUnloadStates.stLockPalletLockFix:
		fixPalletStart := TRUE;	
		io.setSR(ioImage.yPalletFix_lock, ioImage.yPalletFix_unlock);
		nextState(stackerUnloadStates.stLockPalletCheckFix);
		
// *** Lock Pallet - Check Fix
// Проверка дали тарата е фиксирана

	stackerUnloadStates.stLockPalletCheckFix:		
		IF io.getSR(ioImage.xPalletFix_lock, ioImage.xPalletFix_unlock) THEN
		   		nextState(stackerUnloadStates.stLockPalletDone);
		END_IF
		
		IF stateDelay(cylinderTimeOut) THEN
			setError(stackerUnloadStates.stErrFixerNotClose);	
		END_IF		

// *** Lock Pallet - Done

	stackerUnloadStates.stLockPalletDone:
		fixPalletStart := FALSE;
		nextState(stackerUnloadStates.stReady);		

// *** Purge - Start
// Без значение колко палети има те трябва да се извадят от стакера

	stackerUnloadStates.stUnloadPurgeStart:	
		purgeStart := TRUE;
		setDisplayState(stackerUnLoadDisplayStates.dStStackerIsReseting);
		nextState(stackerUnloadStates.stUnloadPurgeCheck);

// *** Purge - Check
// Ако стакера е на долна крайна поз. - се прави Reset

	stackerUnloadStates.stUnloadPurgeCheck:
		IF moveDone AND currentPos = posCount THEN
			nextState(stackerUnloadStates.stUnloadPurgeDone);
		ELSE
			IF Stations.sUnLoadDrive.Enabled AND NOT Stations.sUnLoadDrive.Error THEN
				nextState(stackerUnloadStates.stUnloadPurgeMove);
			 ELSE
				nextState(stackerUnloadStates.stUnloadPurgeDriveOn);
			END_IF	
		END_IF

// *** Purge - Drive On
// Вкл. на инвертора на FESTO мотора на оста на стакера	

	stackerUnloadStates.stUnloadPurgeDriveOn:	
		IF Stations.sUnloadDrive.Error THEN
			Stations.sUnloadDrive.DoReset  := TRUE;
		ELSE
			Stations.sUnloadDrive.DoReset  := FALSE;
			Stations.sUnloadDrive.DoEnable := TRUE;
			IF stateDelay(driveEnTime) THEN
				nextState(stackerUnloadStates.stUnloadPurgeMove);
			END_IF
		END_IF
		timeOutError(driveEnTime*2, stackerUnloadStates.stErrAxis);		
		
// *** Purge - Drive Move
// Прави 1 хода нагоре

	stackerUnloadStates.stUnloadPurgeMove:	
		IF moveDone THEN
			currentPos := currentPos - 1;
		END_IF
		Stations.sUnloadDrive.TargetPosition     := axisPosArr[currentPos];
		Stations.sUnloadDrive.TargetAcceleration := Stations.sUnloadSettings.axisAcc;
		Stations.sUnloadDrive.TargetVelocity     := Stations.sUnloadSettings.axisInitSpeed;
		Stations.sUnloadDrive.DoMove             := TRUE;
		moveDone							     := FALSE;
		IF stateDelay(drivePosTime) THEN		
			nextState(stackerUnloadStates.stUnloadPurgeMoveCheck);
		END_IF	

// *** Purge - Check Drive
// Проверка дали е завършил хода на оста

	stackerUnloadStates.stUnloadPurgeMoveCheck:		
		IF Stations.sUnloadDrive.TargetReached AND NOT Stations.sUnloadDrive.Error THEN
			Stations.sUnloadDrive.DoMove := FALSE;
			moveDone 				     := TRUE;
			nextState(stackerUnloadStates.stUnloadPurgeDone);	
		ELSIF NOT Stations.sUnloadDrive.TargetReached AND Stations.sUnloadDrive.Error THEN
			setError(stackerUnloadStates.stInitMoveErr);
		END_IF	
		timeOutError(palletMoveTimeOut, stackerUnloadStates.stErrPalletMove);			
	
// *** Purge - Done
// От тук стакера се ресетва

	stackerUnloadStates.stUnloadPurgeDone:	
		nextState(stackerUnloadStates.stResetStart);		
		
// *** Step Block State
// В този state се влиза винаги след изпълняването на една стъпка при стъпков режим
	stackerUnloadStates.stStepBlock:
		setDisplayState(stackerUnLoadDisplayStates.dStWaitForNextStep);	
		
// *** Station Stop
// Станцията е била изключена 
 
	stackerUnloadStates.stStop:						   							   
		resetDone			 := FALSE; 		
		prepareDone			 := FALSE;							  
		moveUpStart			 := FALSE;							   
		unlockPalletStart    := FALSE; 						  
		fixPalletStart		 := FALSE; 						  
		purgeStart			 := FALSE; 						   
		moveDone		     := FALSE; 						   						   
	
// Състояния за грешки
	
//  *** ERROR No axis setting
// 	Липсват настойки на оста (ход и размер на тара)	

	stackerUnloadStates.stErrNoProperSettings:
		setDisplayState(stackerUnLoadDisplayStates.dStAxisNotConfigured);

// *** ERROR remove Pallet	
// След старт на машината не трябва да има палет на стакера. 
// Ако има оператора трябва да го махне

	stackerUnloadStates.stErrRemovePallet:
		setDisplayState(stackerUnLoadDisplayStates.dStRemotePalletManually);

// *** ЕRROR  Lock 1 not open
// Цилиндъра не се е отворил навреме
		
	stackerUnloadStates.stErrLock1NotOpen:
		setDisplayState(stackerUnLoadDisplayStates.dStLock1CylinderDidNotOpen);
		
// *** ЕRROR  Lock 1 not close
// Цилиндъра не се е затворил навреме
		
	stackerUnloadStates.stErrLock1NotClose:
		setDisplayState(stackerUnLoadDisplayStates.dStLock1CylinderDidNotClose);	
		
// *** ЕRROR  Lock 2 not open
// Цилиндъра не се е отворил навреме	
	
	stackerUnloadStates.stErrLock2NotOpen:
		setDisplayState(stackerUnLoadDisplayStates.dStLock2CylinderDidNotOpen);		
		
// *** ЕRROR  Lock 2 not close
// Цилиндъра не се е затворил навреме	
	
	stackerUnloadStates.stErrLock2NotClose:
		setDisplayState(stackerUnLoadDisplayStates.dStLock2CylinderDidNotClose);			

// *** ЕRROR  Fixer not open
// Цилиндъра не се е отворил навреме	
	
	stackerUnloadStates.stErrFixerNotOpen:
		setDisplayState(stackerUnLoadDisplayStates.dStFixerCylinderDidNotOpen);	
		
// *** ЕRROR  Fixer not close
// Цилиндъра не се е затворил навреме	
	
	stackerUnloadStates.stErrFixerNotClose:
		setDisplayState(stackerUnLoadDisplayStates.dStFixerCylinderDidNotClose);		

// *** ERROR Axis
// Има грешка на FESTO инвертора

	stackerUnloadStates.stErrAxis:
		Stations.sUnloadDrive.DoEnable     := FALSE;
		setDisplayState(stackerUnLoadDisplayStates.dStFestoDriveError);
		
// ***ERROR Init move
// Движението към горна крайна точка при init е отнело твърде мн. време		
		
	stackerUnloadStates.stInitMoveErr:
		Stations.sUnloadDrive.DoMove       := FALSE;
		Stations.sUnloadDrive.DoEnable     := FALSE;
		setDisplayState(stackerUnLoadDisplayStates.dStAxisInitMoveTakesTooLong);
		
// *** ERROR Pallet Move up
// Движението за преместването на една тара ход нагоре е отнело твърде мн време

	stackerUnloadStates.stErrPalletMove:
		Stations.sUnloadDrive.DoMove       := FALSE;
		Stations.sUnloadDrive.DoEnable     := FALSE;
		setDisplayState(stackerUnLoadDisplayStates.dStPalletMoveTakesTooLong);
		
// *** ERROR Pallet Detected
// На "върха" на стaкера има засечена tara от xPalletOnTop, а не трябва
// Вероятно проблем със самият сензор
	
	stackerUnloadStates.stErrPalletDetected:
		setDisplayState(stackerUnLoadDisplayStates.dStPalletIsDetectedFault);

// *** ERROR No Pallet
// Стакер се опитва да зареди тари, но не открива тара на върха

	stackerUnloadStates.stErrNoPallet:
		setDisplayState(stackerUnLoadDisplayStates.dStThereIsNoPalletOnTop);		
		
// *** EMG Stop
// Аварийно спиране при натискане на гъба или отваряне на врата

	stackerUnloadStates.stEMG:	
		
		Stations.sUnloadDrive.DoMove       := FALSE;
		Stations.sUnloadDrive.DoEnable     := FALSE;
		
		nextState(stackerUnloadStates.stInit);
	
END_CASE

ACTION drivesControl:


axisFesto          ( axis				:= Stations.sUnloadAxis,
					PowerUP 			:= Stations.sUnloadDrive.DoEnable, 
					Home 				:= Stations.sUnloadDrive.DoHome, 
					StartMove 			:= Stations.sUnloadDrive.DoMove, 
					Reset 				:= Stations.sUnloadDrive.DoReset, 
					Position 			:= Stations.sUnloadDrive.TargetPosition, 
					Velocity 			:= Stations.sUnloadDrive.TargetVelocity,
					Acceleration		:= Stations.sUnloadDrive.TargetAcceleration,
					IsAbsolute 			:= TRUE,
					Enabled 			=> Stations.sUnloadDrive.Enabled,
					Error 				=> Stations.sUnloadDrive.Error,
					ErrorID 			=> Stations.sUnloadDrive.ErrorID,
					TargetReached 		=> Stations.sUnloadDrive.TargetReached,
					HomeDone 			=> Stations.sUnloadDrive.Refferenced,
					Moving 				=> Stations.sUnloadDrive.Moving,
					CurrentPosition 	=> Stations.sUnloadDrive.CurrentPosition,
					OperationMode		=> Stations.sUnloadDrive.OperationMode);
END_ACTION

END_FUNCTION_BLOCK

// ---- POUs/Stations/insertLoadStation.TcPOU
FUNCTION_BLOCK insertLoadStation EXTENDS stateMachine
VAR_INPUT
	
	ioImage                : inserterLoadImage;

END_VAR

VAR

	activeState            : inserterLoadStates;	
	axisLinMot             : FB_ServoAxis_LinMot; 
	
	resetDone			   : BOOL := FALSE; 						   // Инсъртъра е ресетнат
	prepareStart           : BOOL := FALSE; 						   // Изчаква синхронизация с индекс масата
	loadStart              : BOOL := FALSE; 						   // Робота е донесъл нов сензор
	rotStart               : BOOL := FALSE; 						   // Начално поз. на ротатора
	posStart               : BOOL := FALSE; 						   // Ротира сензора на позиция, спрямо команда от камерата
	insertStart            : BOOL := FALSE;							   // Поставяне на сензора в гнездото на масата
	releaseStart           : BOOL := FALSE; 						   // Връщане на инсъртъра в начлана поз.
	syncStart			   : BOOL := FALSE; 						   // Sync с индекс масата, че работа е завършена

	
	initRotPos			   : REAL; 									   // Начално завъртане
	camRotPos              : REAL;                                     // Завъртане за снимка
	workRotPos             : REAL;                                     // Завъртане след снимка - cw ии ccw
	cwRotPos               : REAL;
    ccwRotPos              : REAL;                                      
	
